# B&R Automation Studio project OpcUaSample410_BrbLibUa103 (part 13)

#### BrbUaRcGetNodeHandle.c
```c
#include <bur/plctypes.h>
#ifdef __cplusplus
	extern "C"
	{
#endif

#include "BrbLibUa.h"
#include <string.h>
#include <AnsiCFunc.h>

#ifdef __cplusplus
	};
#endif

// NOLINTBEGIN(readability-*, bugprone-easily-swappable-parameters, bugprone-branch-clone, clang-diagnostic-invalid-utf8, clang-diagnostic-invalid-source-encoding, clang-diagnostic-pointer-arith, clang-diagnostic-strict-prototypes, hicpp-uppercase-literal-suffix, cppcoreguidelines-*, performance-*)

/* Gibt einen ermittelten NodeHandle zurück */
unsigned short BrbUaRcGetNodeHandle(struct BrbUaRunClient_TYP* pRunClient, unsigned short nNodeHandleIndex, struct BrbUaRcNodeHandle_TYP* pNodeHandle)
{
	UINT nStatus = eBRB_ERR_NULL_POINTER;
	if(pRunClient != 0 && pNodeHandle != 0)
	{
		memset(pNodeHandle, 0, sizeof(BrbUaRcNodeHandle_TYP));
		nStatus = eBRB_ERR_UA_NO_ELEMENTS;
		if(pRunClient->NodeHandles.nNodeHandleCount > 0 && pRunClient->NodeHandles.pDatObjNamespaceIndices != 0 && pRunClient->NodeHandles.pNodeIds != 0 && pRunClient->NodeHandles.pNodeHandleErrorIds != 0 && pRunClient->NodeHandles.pNodeHandles != 0)
		{
			nStatus = eBRB_ERR_UA_INVALID_INDEX;
			if(nNodeHandleIndex < pRunClient->NodeHandles.nNodeHandleCount)
			{
				nStatus = eBRB_ERR_OK;
				pNodeHandle->nDatObjNamespaceIndex = *(((UINT*)pRunClient->NodeHandles.pDatObjNamespaceIndices) + nNodeHandleIndex);
				memcpy(&pNodeHandle->NodeId, (USINT*)(((UANodeID*)pRunClient->NodeHandles.pNodeIds) + nNodeHandleIndex), sizeof(UANodeID));
				pNodeHandle->nErrorId = *(((DWORD*)pRunClient->NodeHandles.pNodeHandleErrorIds) + nNodeHandleIndex);
				pNodeHandle->nNodeHandle = *(((DWORD*)pRunClient->NodeHandles.pNodeHandles) + nNodeHandleIndex);
			}
		}
	}
	return nStatus;
}

// NOLINTEND(readability-*, bugprone-easily-swappable-parameters, bugprone-branch-clone, clang-diagnostic-invalid-utf8, clang-diagnostic-invalid-source-encoding, clang-diagnostic-pointer-arith, clang-diagnostic-strict-prototypes, hicpp-uppercase-literal-suffix, cppcoreguidelines-*, performance-*)
```

#### BrbUaRcGetReadBlock.c
```c
#include <bur/plctypes.h>
#ifdef __cplusplus
	extern "C"
	{
#endif

#include "BrbLibUa.h"
#include <string.h>
#include <AnsiCFunc.h>

#ifdef __cplusplus
	};
#endif

// NOLINTBEGIN(readability-*, bugprone-easily-swappable-parameters, bugprone-branch-clone, clang-diagnostic-invalid-utf8, clang-diagnostic-invalid-source-encoding, clang-diagnostic-pointer-arith, clang-diagnostic-strict-prototypes, hicpp-uppercase-literal-suffix, cppcoreguidelines-*, performance-*)

/* Gibt einen ermittelten ReadBlock zurück */
unsigned short BrbUaRcGetReadBlock(struct BrbUaRunClient_TYP* pRunClient, unsigned short nReadBlockIndex, struct BrbUaRcReadBlock_TYP* pReadBlock, struct BrbUaRcReadBlockIntern_TYP* pReadBlockIntern)
{
	UINT nStatus = eBRB_ERR_NULL_POINTER;
	if(pRunClient != 0 && pReadBlock != 0)
	{
		memset(pReadBlock, 0, sizeof(BrbUaRcReadBlock_TYP));
		nStatus = eBRB_ERR_UA_NO_ELEMENTS;
		if(pRunClient->ReadBlocks.nBlockCount > 0 && pRunClient->ReadBlocks.pBlocks != 0)
		{
			nStatus = eBRB_ERR_UA_INVALID_INDEX;
			if(nReadBlockIndex < pRunClient->ReadBlocks.nBlockCount)
			{
				nStatus = eBRB_ERR_OK;
				BrbUaRcReadBlockIntern_TYP* pReadBlockInternOri = ((BrbUaRcReadBlockIntern_TYP*)pRunClient->ReadBlocks.pBlocks) + nReadBlockIndex;
				pReadBlock->nReadItemCount = pReadBlockInternOri->nReadItemCount;
				if(pReadBlockIntern != 0)
				{
					memcpy(pReadBlockIntern, pReadBlockInternOri, sizeof(BrbUaRcReadBlockIntern_TYP));
				}
			}
		}
	}
	return nStatus;
}

// NOLINTEND(readability-*, bugprone-easily-swappable-parameters, bugprone-branch-clone, clang-diagnostic-invalid-utf8, clang-diagnostic-invalid-source-encoding, clang-diagnostic-pointer-arith, clang-diagnostic-strict-prototypes, hicpp-uppercase-literal-suffix, cppcoreguidelines-*, performance-*)
```

#### BrbUaRcGetReadItem.c
```c
#include <bur/plctypes.h>
#ifdef __cplusplus
	extern "C"
	{
#endif

#include "BrbLibUa.h"
#include <string.h>
#include <AnsiCFunc.h>

#ifdef __cplusplus
	};
#endif

// NOLINTBEGIN(readability-*, bugprone-easily-swappable-parameters, bugprone-branch-clone, clang-diagnostic-invalid-utf8, clang-diagnostic-invalid-source-encoding, clang-diagnostic-pointer-arith, clang-diagnostic-strict-prototypes, hicpp-uppercase-literal-suffix, cppcoreguidelines-*, performance-*)

/* Gibt ein ermitteltes ReadItem zurück */
unsigned short BrbUaRcGetReadItem(struct BrbUaRunClient_TYP* pRunClient, unsigned short nReadBlockIndex, unsigned short nReadItemIndex, struct BrbUaRcReadItem_TYP* pReadItem)
{
	UINT nStatus = eBRB_ERR_NULL_POINTER;
	if(pRunClient != 0 && pReadItem != 0)
	{
		memset(pReadItem, 0, sizeof(BrbUaRcReadItem_TYP));
		nStatus = eBRB_ERR_UA_NO_ELEMENTS;
		if(pRunClient->ReadBlocks.nBlockCount > 0 && pRunClient->ReadBlocks.pBlocks != 0)
		{
			nStatus = eBRB_ERR_UA_INVALID_INDEX;
			if(nReadBlockIndex < pRunClient->ReadBlocks.nBlockCount)
			{
				nStatus = eBRB_ERR_UA_NO_ELEMENTS;
				BrbUaRcReadBlockIntern_TYP* pReadBlock = ((BrbUaRcReadBlockIntern_TYP*)pRunClient->ReadBlocks.pBlocks) + nReadBlockIndex;
				if(pReadBlock->nReadItemCount > 0 &&
					pReadBlock->pRiDatObjNamespaceIndices != 0 && pReadBlock->pRiNodeIds != 0 &&
					pReadBlock->pRiNodeAddInfos != 0 && pReadBlock->pRiVariables != 0 &&
					pReadBlock->pRiNodeErrorIds != 0 && pReadBlock->pRiTimestamps != 0
					)
				{
					nStatus = eBRB_ERR_UA_INVALID_INDEX;
					if(nReadItemIndex < pReadBlock->nReadItemCount)
					{
						nStatus = eBRB_ERR_OK;
						pReadItem->nDatObjNamespaceIndex = *(((UINT*)pReadBlock->pRiDatObjNamespaceIndices) + nReadItemIndex);
						memcpy(&pReadItem->NodeId, ((UANodeID*)pReadBlock->pRiNodeIds) + nReadItemIndex, sizeof(UANodeID));
						UANodeAdditionalInfo* pNodeAddInfo = ((UANodeAdditionalInfo*)pReadBlock->pRiNodeAddInfos) + nReadItemIndex;
						memcpy(&pReadItem->AddInfo, pNodeAddInfo, sizeof(UANodeAdditionalInfo));
						STRING sVarName[nBRBUA_VARNAME_TEXT_CHAR_MAX+1];
						STRING* pVar = (STRING*)((USINT*)pReadBlock->pRiVariables) + (nReadItemIndex * sizeof(sVarName));
						BrbStringCopy(pReadItem->sVar, pVar, sizeof(pReadItem->sVar));
						pReadItem->dtTimestamp = *(((DATE_AND_TIME*)pReadBlock->pRiTimestamps) + nReadItemIndex);
						pReadItem->nErrorId = *(((DWORD*)pReadBlock->pRiNodeErrorIds) + nReadItemIndex);
					}
				}
			}
		}
	}
	return nStatus;
}

// NOLINTEND(readability-*, bugprone-easily-swappable-parameters, bugprone-branch-clone, clang-diagnostic-invalid-utf8, clang-diagnostic-invalid-source-encoding, clang-diagnostic-pointer-arith, clang-diagnostic-strict-prototypes, hicpp-uppercase-literal-suffix, cppcoreguidelines-*, performance-*)
```

#### BrbUaRcGetWriteBlock.c
```c
#include <bur/plctypes.h>
#ifdef __cplusplus
	extern "C"
	{
#endif

#include "BrbLibUa.h"
#include <string.h>
#include <AnsiCFunc.h>

#ifdef __cplusplus
	};
#endif

// NOLINTBEGIN(readability-*, bugprone-easily-swappable-parameters, bugprone-branch-clone, clang-diagnostic-invalid-utf8, clang-diagnostic-invalid-source-encoding, clang-diagnostic-pointer-arith, clang-diagnostic-strict-prototypes, hicpp-uppercase-literal-suffix, cppcoreguidelines-*, performance-*)

/* Gibt einen ermittelten WriteBlock zurück */
unsigned short BrbUaRcGetWriteBlock(struct BrbUaRunClient_TYP* pRunClient, unsigned short nWriteBlockIndex, struct BrbUaRcWriteBlock_TYP* pWriteBlock, struct BrbUaRcWriteBlockIntern_TYP* pWriteBlockIntern)
{
	UINT nStatus = eBRB_ERR_NULL_POINTER;
	if(pRunClient != 0 && pWriteBlock != 0)
	{
		memset(pWriteBlock, 0, sizeof(BrbUaRcWriteBlock_TYP));
		nStatus = eBRB_ERR_UA_NO_ELEMENTS;
		if(pRunClient->WriteBlocks.nBlockCount > 0 && pRunClient->WriteBlocks.pBlocks != 0)
		{
			nStatus = eBRB_ERR_UA_INVALID_INDEX;
			if(nWriteBlockIndex < pRunClient->WriteBlocks.nBlockCount)
			{
				nStatus = eBRB_ERR_OK;
				BrbUaRcWriteBlockIntern_TYP* pWriteBlockInternOri = ((BrbUaRcWriteBlockIntern_TYP*)pRunClient->WriteBlocks.pBlocks) + nWriteBlockIndex;
				pWriteBlock->nWriteItemCount = pWriteBlockInternOri->nWriteItemCount;
				if(pWriteBlockIntern != 0)
				{
					memcpy(pWriteBlockIntern, pWriteBlockInternOri, sizeof(BrbUaRcWriteBlockIntern_TYP));
				}
			}
		}
	}
	return nStatus;
}

// NOLINTEND(readability-*, bugprone-easily-swappable-parameters, bugprone-branch-clone, clang-diagnostic-invalid-utf8, clang-diagnostic-invalid-source-encoding, clang-diagnostic-pointer-arith, clang-diagnostic-strict-prototypes, hicpp-uppercase-literal-suffix, cppcoreguidelines-*, performance-*)
```

#### BrbUaRcGetWriteItem.c
```c
#include <bur/plctypes.h>
#ifdef __cplusplus
	extern "C"
	{
#endif

#include "BrbLibUa.h"
#include <string.h>
#include <AnsiCFunc.h>

#ifdef __cplusplus
	};
#endif

// NOLINTBEGIN(readability-*, bugprone-easily-swappable-parameters, bugprone-branch-clone, clang-diagnostic-invalid-utf8, clang-diagnostic-invalid-source-encoding, clang-diagnostic-pointer-arith, clang-diagnostic-strict-prototypes, hicpp-uppercase-literal-suffix, cppcoreguidelines-*, performance-*)

/* Gibt ein ermitteltes WriteItem zurück */
unsigned short BrbUaRcGetWriteItem(struct BrbUaRunClient_TYP* pRunClient, unsigned short nWriteBlockIndex, unsigned short nWriteItemIndex, struct BrbUaRcWriteItem_TYP* pWriteItem)
{
	UINT nStatus = eBRB_ERR_NULL_POINTER;
	if(pRunClient != 0 && pWriteItem != 0)
	{
		memset(pWriteItem, 0, sizeof(BrbUaRcWriteItem_TYP));
		nStatus = eBRB_ERR_UA_NO_ELEMENTS;
		if(pRunClient->WriteBlocks.nBlockCount > 0 && pRunClient->WriteBlocks.pBlocks != 0)
		{
			nStatus = eBRB_ERR_UA_INVALID_INDEX;
			if(nWriteBlockIndex < pRunClient->WriteBlocks.nBlockCount)
			{
				nStatus = eBRB_ERR_UA_NO_ELEMENTS;
				BrbUaRcWriteBlockIntern_TYP* pWriteBlock = ((BrbUaRcWriteBlockIntern_TYP*)pRunClient->WriteBlocks.pBlocks) + nWriteBlockIndex;
				if(pWriteBlock->nWriteItemCount > 0 &&
					pWriteBlock->pWiDatObjNamespaceIndices != 0 && pWriteBlock->pWiNodeIds != 0 &&
					pWriteBlock->pWiNodeAddInfos != 0 && pWriteBlock->pWiVariables != 0 &&
					pWriteBlock->pWiNodeErrorIds != 0
					)
				{
					nStatus = eBRB_ERR_UA_INVALID_INDEX;
					if(nWriteItemIndex < pWriteBlock->nWriteItemCount)
					{
						nStatus = eBRB_ERR_OK;
						pWriteItem->nDatObjNamespaceIndex = *(((UINT*)pWriteBlock->pWiDatObjNamespaceIndices) + nWriteItemIndex);
						memcpy(&pWriteItem->NodeId, ((UANodeID*)pWriteBlock->pWiNodeIds) + nWriteItemIndex, sizeof(UANodeID));
						UANodeAdditionalInfo* pNodeAddInfo = ((UANodeAdditionalInfo*)pWriteBlock->pWiNodeAddInfos) + nWriteItemIndex;
						memcpy(&pWriteItem->AddInfo, pNodeAddInfo, sizeof(UANodeAdditionalInfo));
						STRING sVarName[nBRBUA_VARNAME_TEXT_CHAR_MAX+1];
						STRING* pVar = (STRING*)((USINT*)pWriteBlock->pWiVariables) + (nWriteItemIndex * sizeof(sVarName));
						BrbStringCopy(pWriteItem->sVar, pVar, sizeof(pWriteItem->sVar));
						pWriteItem->nErrorId = *(((DWORD*)pWriteBlock->pWiNodeErrorIds) + nWriteItemIndex);
					}
				}
			}
		}
	}
	return nStatus;
}

// NOLINTEND(readability-*, bugprone-easily-swappable-parameters, bugprone-branch-clone, clang-diagnostic-invalid-utf8, clang-diagnostic-invalid-source-encoding, clang-diagnostic-pointer-arith, clang-diagnostic-strict-prototypes, hicpp-uppercase-literal-suffix, cppcoreguidelines-*, performance-*)
```

#### BrbUaRcGetMethod.c
```c
#include <bur/plctypes.h>
#ifdef __cplusplus
	extern "C"
	{
#endif

#include "BrbLibUa.h"
#include <string.h>
#include <AnsiCFunc.h>

#ifdef __cplusplus
	};
#endif

// NOLINTBEGIN(readability-*, bugprone-easily-swappable-parameters, bugprone-branch-clone, clang-diagnostic-invalid-utf8, clang-diagnostic-invalid-source-encoding, clang-diagnostic-pointer-arith, clang-diagnostic-strict-prototypes, hicpp-uppercase-literal-suffix, cppcoreguidelines-*, performance-*)

/* Gibt eine ermittelte Methode zuück */
unsigned short BrbUaRcGetMethod(struct BrbUaRunClient_TYP* pRunClient, unsigned short nMethodIndex, struct BrbUaRcMethod_TYP* pMethod, struct BrbUaRcMethodIntern_TYP* pMethodIntern)
{
	UINT nStatus = eBRB_ERR_NULL_POINTER;
	if(pRunClient != 0 && pMethod != 0)
	{
		memset(pMethod, 0, sizeof(BrbUaRcMethod_TYP));
		nStatus = eBRB_ERR_UA_NO_ELEMENTS;
		if(pRunClient->Methods.nMethodCount > 0 && pRunClient->Methods.pMethods != 0)
		{
			nStatus = eBRB_ERR_UA_INVALID_INDEX;
			if(nMethodIndex < pRunClient->Methods.nMethodCount)
			{
				nStatus = eBRB_ERR_OK;
				BrbUaRcMethodIntern_TYP* pMethodInternOri = (((BrbUaRcMethodIntern_TYP*)pRunClient->Methods.pMethods)  + nMethodIndex);
				pMethod->nDatObjNamespaceIndex = pMethodInternOri->nDatObjNamespaceIndex;
				memcpy(&pMethod->ObjectNodeId, &pMethodInternOri->ObjectNodeId, sizeof(UANodeID));
				memcpy(&pMethod->MethodNodeId, &pMethodInternOri->MethodNodeId, sizeof(UANodeID));
				pMethod->tTimeout = pMethodInternOri->tTimeout;
				pMethod->nInputArgsCount = pMethodInternOri->nInputArgsCount;
				pMethod->nOutputArgsCount = pMethodInternOri->nOutputArgsCount;
				pMethod->nErrorId = pMethodInternOri->nErrorId;
				pMethod->nMethodHandle = pMethodInternOri->nMethodHandle;
				if(pMethodIntern != 0)
				{
					memcpy(pMethodIntern, pMethodInternOri, sizeof(BrbUaRcMethodIntern_TYP));
				}
			}
		}
	}
	return nStatus;
}

// NOLINTEND(readability-*, bugprone-easily-swappable-parameters, bugprone-branch-clone, clang-diagnostic-invalid-utf8, clang-diagnostic-invalid-source-encoding, clang-diagnostic-pointer-arith, clang-diagnostic-strict-prototypes, hicpp-uppercase-literal-suffix, cppcoreguidelines-*, performance-*)
```

#### BrbUaRcGetArgument.c
```c
#include <bur/plctypes.h>
#ifdef __cplusplus
	extern "C"
	{
#endif

#include "BrbLibUa.h"
#include <string.h>
#include <AnsiCFunc.h>

#ifdef __cplusplus
	};
#endif

// NOLINTBEGIN(readability-*, bugprone-easily-swappable-parameters, bugprone-branch-clone, clang-diagnostic-invalid-utf8, clang-diagnostic-invalid-source-encoding, clang-diagnostic-pointer-arith, clang-diagnostic-strict-prototypes, hicpp-uppercase-literal-suffix, cppcoreguidelines-*, performance-*)

/* Gibt ein ermitteltes ReadItem zurück */
unsigned short BrbUaRcGetArgument(struct BrbUaRunClient_TYP* pRunClient, unsigned short nMethodIndex, plcbit bOutput, unsigned short nArgumentIndex, struct UAMethodArgument* pArgument)
{
	UINT nStatus = eBRB_ERR_NULL_POINTER;
	if(pRunClient != 0 && pArgument != 0)
	{
		memset(pArgument, 0, sizeof(UAMethodArgument));
		nStatus = eBRB_ERR_UA_NO_ELEMENTS;
		if(pRunClient->Methods.nMethodCount > 0 && pRunClient->Methods.pMethods != 0)
		{
			nStatus = eBRB_ERR_UA_INVALID_INDEX;
			if(nMethodIndex < pRunClient->Methods.nMethodCount)
			{
				nStatus = eBRB_ERR_UA_NO_ELEMENTS;
				BrbUaRcMethodIntern_TYP* pMethod = (((BrbUaRcMethodIntern_TYP*)pRunClient->Methods.pMethods) + nMethodIndex);
				if(bOutput == 0)
				{
					if(pMethod->nInputArgsCount > 0 && pMethod->pInputArguments != 0)
					{
						nStatus = eBRB_ERR_UA_INVALID_INDEX;
						if(nArgumentIndex < pMethod->nInputArgsCount)
						{
							nStatus = eBRB_ERR_OK;
							UAMethodArgument* pArgumentIntern = ((UAMethodArgument*)pMethod->pInputArguments) + nArgumentIndex;
							memcpy(pArgument, pArgumentIntern, sizeof(UAMethodArgument));
						}
					}
				}
				else
				{
					if(pMethod->nOutputArgsCount > 0 && pMethod->pOutputArguments != 0)
					{
						nStatus = eBRB_ERR_UA_INVALID_INDEX;
						if(nArgumentIndex < pMethod->nOutputArgsCount)
						{
							nStatus = eBRB_ERR_OK;
							UAMethodArgument* pArgumentIntern = ((UAMethodArgument*)pMethod->pOutputArguments) + nArgumentIndex;
							memcpy(pArgument, pArgumentIntern, sizeof(UAMethodArgument));
						}
					}
				}
			}
		}
	}
	return nStatus;
}

// NOLINTEND(readability-*, bugprone-easily-swappable-parameters, bugprone-branch-clone, clang-diagnostic-invalid-utf8, clang-diagnostic-invalid-source-encoding, clang-diagnostic-pointer-arith, clang-diagnostic-strict-prototypes, hicpp-uppercase-literal-suffix, cppcoreguidelines-*, performance-*)
```

#### BrbUaRcGetSubscription.c
```c
#include <bur/plctypes.h>
#ifdef __cplusplus
	extern "C"
	{
#endif

#include "BrbLibUa.h"
#include <string.h>
#include <AnsiCFunc.h>

#ifdef __cplusplus
	};
#endif

// NOLINTBEGIN(readability-*, bugprone-easily-swappable-parameters, bugprone-branch-clone, clang-diagnostic-invalid-utf8, clang-diagnostic-invalid-source-encoding, clang-diagnostic-pointer-arith, clang-diagnostic-strict-prototypes, hicpp-uppercase-literal-suffix, cppcoreguidelines-*, performance-*)

/* Gibt eine ermittelte Subscription zurück */
unsigned short BrbUaRcGetSubscription(struct BrbUaRunClient_TYP* pRunClient, unsigned short nSubscriptionIndex, struct BrbUaRcSubscription_TYP* pSubscription, struct BrbUaRcSubscriptionIntern_TYP* pSubscriptionIntern)
{
	UINT nStatus = eBRB_ERR_NULL_POINTER;
	if(pRunClient != 0 && pSubscription != 0)
	{
		memset(pSubscription, 0, sizeof(BrbUaRcSubscription_TYP));
		nStatus = eBRB_ERR_UA_NO_ELEMENTS;
		if(pRunClient->Subscriptions.nSubscriptionCount > 0 && pRunClient->Subscriptions.pSubscriptions != 0)
		{
			nStatus = eBRB_ERR_UA_INVALID_INDEX;
			if(nSubscriptionIndex < pRunClient->Subscriptions.nSubscriptionCount)
			{
				nStatus = eBRB_ERR_OK;
				BrbUaRcSubscriptionIntern_TYP* pSubscriptionInternOri = ((BrbUaRcSubscriptionIntern_TYP*)pRunClient->Subscriptions.pSubscriptions) + nSubscriptionIndex;
				pSubscription->bPublishingEnable = pSubscriptionInternOri->bPublishingEnable;
				pSubscription->nPriority = pSubscriptionInternOri->nPriority;
				pSubscription->tPublishingInterval = pSubscriptionInternOri->tPublishingInterval;
				pSubscription->nMonitoredItemCount = pSubscriptionInternOri->nMonitoredItemCount;
				pSubscription->nEventItemCount = pSubscriptionInternOri->nEventItemCount;
				pSubscription->nErrorId = pSubscriptionInternOri->nErrorId;
				pSubscription->nSubscriptionHandle = pSubscriptionInternOri->nSubscriptionHandle;
				if(pSubscriptionIntern != 0)
				{
					memcpy(pSubscriptionIntern, pSubscriptionInternOri, sizeof(BrbUaRcSubscriptionIntern_TYP));
				}
			}
		}
	}
	return nStatus;
}

// NOLINTEND(readability-*, bugprone-easily-swappable-parameters, bugprone-branch-clone, clang-diagnostic-invalid-utf8, clang-diagnostic-invalid-source-encoding, clang-diagnostic-pointer-arith, clang-diagnostic-strict-prototypes, hicpp-uppercase-literal-suffix, cppcoreguidelines-*, performance-*)
```

#### BrbUaRcSetSubscription.c
```c
#include <bur/plctypes.h>
#ifdef __cplusplus
	extern "C"
	{
#endif

#include "BrbLibUa.h"
#include <string.h>
#include <AnsiCFunc.h>

#ifdef __cplusplus
	};
#endif

// NOLINTBEGIN(readability-*, bugprone-easily-swappable-parameters, bugprone-branch-clone, clang-diagnostic-invalid-utf8, clang-diagnostic-invalid-source-encoding, clang-diagnostic-pointer-arith, clang-diagnostic-strict-prototypes, hicpp-uppercase-literal-suffix, cppcoreguidelines-*, performance-*)

// Eigene Enums und Typen
enum Steps_ENUM
{
	eSTEP_INIT,
	eSTEP_OPERATE,
	eSTEP_OPERATE_WAIT,
};

/* Ändert die Parameter einer Subscription */
void BrbUaRcSetSubscription(struct BrbUaRcSetSubscription* inst)
{
	switch(inst->eStep)
	{
		case eSTEP_INIT:
			// Fub initialisieren
			inst->nStatus =  eBRB_ERR_BUSY;
			inst->bPublished = 0;
			inst->nErrorId = 0x00000000; // Good
			BrbUaGetStatusCodeText(inst->nErrorId, inst->sErrorId, sizeof(inst->nErrorId));
			memset(&inst->fbUA_SubscriptionOperate, 0, sizeof(inst->fbUA_SubscriptionOperate));
			// Parameter prüfen
			if(inst->pRunClient != 0 && inst->pSubscription != 0)
			{
				if(inst->pRunClient->State.eClientState == eBRB_RCCLTSTATE_CONNECTED && inst->pRunClient->Connection.nConnectionHandle != 0)
				{
					if(inst->pRunClient->Subscriptions.nSubscriptionCount > 0 && inst->pRunClient->Subscriptions.pSubscriptions != 0)
					{
						if(inst->nSubscriptionIndex < inst->pRunClient->Subscriptions.nSubscriptionCount)
						{
							inst->eStep = eSTEP_OPERATE;
						}
						else
						{
							inst->nStatus = eBRB_ERR_UA_INVALID_INDEX;
						}
					}
					else
					{
						inst->nStatus = eBRB_ERR_UA_NO_ELEMENTS;
					}
				}
				else
				{
					inst->nStatus = eBRB_ERR_UA_NOT_CONNECTED;
				}
			}
			else
			{
				inst->nStatus = eBRB_ERR_NULL_POINTER;
			}
			break;

		case eSTEP_OPERATE:
			// Subscription ändern
			inst->nStatus  = eBRB_ERR_BUSY;
			{
				BrbUaRcSubscriptionIntern_TYP* pSubscriptionIntern = ((BrbUaRcSubscriptionIntern_TYP*)inst->pRunClient->Subscriptions.pSubscriptions) + inst->nSubscriptionIndex;
				inst->fbUA_SubscriptionOperate.Execute = 1;
				inst->fbUA_SubscriptionOperate.SubscriptionHdl = pSubscriptionIntern->nSubscriptionHandle;
				inst->fbUA_SubscriptionOperate.PublishingEnable = inst->pSubscription->bPublishingEnable;
				inst->fbUA_SubscriptionOperate.Priority = inst->pSubscription->nPriority;
				inst->fbUA_SubscriptionOperate.Timeout = inst->pRunClient->Cfg.tAccessTimeout;
				inst->tPublishingInterval = inst->pSubscription->tPublishingInterval;
				inst->fbUA_SubscriptionOperate.PublishingInterval = &inst->tPublishingInterval;
			}
			inst->eStep = eSTEP_OPERATE_WAIT;
			break;

		case eSTEP_OPERATE_WAIT:
			// Warten, bis Subscription geändert wurde
			inst->nStatus  = eBRB_ERR_BUSY;
			if(inst->fbUA_SubscriptionOperate.Done == 1)
			{
				inst->fbUA_SubscriptionOperate.Execute = 0;
				// Geänderte Werte in interne Daten übernehmen
				BrbUaRcSubscriptionIntern_TYP* pSubscriptionIntern = ((BrbUaRcSubscriptionIntern_TYP*)inst->pRunClient->Subscriptions.pSubscriptions) + inst->nSubscriptionIndex;
				pSubscriptionIntern->bPublishingEnable = inst->pSubscription->bPublishingEnable;
				pSubscriptionIntern->nPriority = inst->pSubscription->nPriority;
				pSubscriptionIntern->tPublishingInterval = inst->pSubscription->tPublishingInterval = inst->tPublishingInterval;
				inst->nStatus  = eBRB_ERR_OK;
				inst->bPublished = inst->fbUA_SubscriptionOperate.Published;
				inst->nErrorId = inst->fbUA_SubscriptionOperate.ErrorID;
				BrbUaGetStatusCodeText(inst->nErrorId, inst->sErrorId, sizeof(inst->nErrorId));
				inst->eStep = eSTEP_INIT;
			}
			else if(inst->fbUA_SubscriptionOperate.Error == 1)
			{
				inst->fbUA_SubscriptionOperate.Execute = 0;
				inst->nStatus  = eBRB_ERR_UA_ERROR;
				inst->nErrorId = inst->fbUA_SubscriptionOperate.ErrorID;
				BrbUaGetStatusCodeText(inst->nErrorId, inst->sErrorId, sizeof(inst->nErrorId));
				inst->eStep = eSTEP_INIT;
			}
			break;

	}

	// Aufruf aller FB's
	UA_SubscriptionOperate(&inst->fbUA_SubscriptionOperate);

}

// NOLINTEND(readability-*, bugprone-easily-swappable-parameters, bugprone-branch-clone, clang-diagnostic-invalid-utf8, clang-diagnostic-invalid-source-encoding, clang-diagnostic-pointer-arith, clang-diagnostic-strict-prototypes, hicpp-uppercase-literal-suffix, cppcoreguidelines-*, performance-*)
```

#### BrbUaRcGetMonitoredItem.c
```c
#include <bur/plctypes.h>
#ifdef __cplusplus
	extern "C"
	{
#endif

#include "BrbLibUa.h"
#include <string.h>
#include <AnsiCFunc.h>

#ifdef __cplusplus
	};
#endif

// NOLINTBEGIN(readability-*, bugprone-easily-swappable-parameters, bugprone-branch-clone, clang-diagnostic-invalid-utf8, clang-diagnostic-invalid-source-encoding, clang-diagnostic-pointer-arith, clang-diagnostic-strict-prototypes, hicpp-uppercase-literal-suffix, cppcoreguidelines-*, performance-*)

/* Gibt ein ermitteltes MonitoredItem zurück */
unsigned short BrbUaRcGetMonitoredItem(struct BrbUaRunClient_TYP* pRunClient, unsigned short nSubscriptionIndex, unsigned short nMonitoredItemIndex, struct BrbUaRcMonitoredItem_TYP* pMonitoredItem)
{
	UINT nStatus = eBRB_ERR_NULL_POINTER;
	if(pRunClient != 0 && pMonitoredItem != 0)
	{
		memset(pMonitoredItem, 0, sizeof(BrbUaRcMonitoredItem_TYP));
		nStatus = eBRB_ERR_UA_NO_ELEMENTS;
		if(pRunClient->Subscriptions.nSubscriptionCount > 0 && pRunClient->Subscriptions.pSubscriptions != 0)
		{
			nStatus = eBRB_ERR_UA_INVALID_INDEX;
			if(nSubscriptionIndex < pRunClient->Subscriptions.nSubscriptionCount)
			{
				nStatus = eBRB_ERR_UA_NO_ELEMENTS;
				BrbUaRcSubscriptionIntern_TYP* pSubscription = ((BrbUaRcSubscriptionIntern_TYP*)pRunClient->Subscriptions.pSubscriptions) + nSubscriptionIndex;
				if(pSubscription->nMonitoredItemCount > 0 &&
					pSubscription->pMiDatObjNamespaceIndices != 0 && pSubscription->pMiNodeIds != 0 &&
					pSubscription->pMiNodeHandleErrorIds != 0 && pSubscription->pMiNodeHandles != 0 &&
					pSubscription->pMiNodeAddInfos != 0 && pSubscription->pMiVariables != 0 &&
					pSubscription->pMiQueueSizeOri != 0 && pSubscription->pMiMonitorSettings != 0 &&
					pSubscription->pMiValuesChanged != 0 && pSubscription->pMiRemainingValueCounts != 0 &&
					pSubscription->pMiTimestamps != 0 && pSubscription->pMiNodeQualityIds != 0 &&
					pSubscription->pMiMonitoredItemErrorIds != 0 && pSubscription->pMiMonitoredItemHandles != 0
					)
				{
					nStatus = eBRB_ERR_UA_INVALID_INDEX;
					if(nMonitoredItemIndex < pSubscription->nMonitoredItemCount)
					{
						nStatus = eBRB_ERR_OK;
						pMonitoredItem->nDatObjNamespaceIndex = *(((UINT*)pSubscription->pMiDatObjNamespaceIndices) + nMonitoredItemIndex);
						memcpy(&pMonitoredItem->NodeId, ((UANodeID*)pSubscription->pMiNodeIds) + nMonitoredItemIndex, sizeof(UANodeID));
						pMonitoredItem->nNodeHandleErrorId = *(((DWORD*)pSubscription->pMiNodeHandleErrorIds) + nMonitoredItemIndex);
						pMonitoredItem->nNodeHandle = *(((DWORD*)pSubscription->pMiNodeHandles) + nMonitoredItemIndex);
						UANodeAdditionalInfo* pNodeAddInfo = ((UANodeAdditionalInfo*)pSubscription->pMiNodeAddInfos) + nMonitoredItemIndex;
						memcpy(&pMonitoredItem->AddInfo, pNodeAddInfo, sizeof(UANodeAdditionalInfo));
						STRING sVarName[nBRBUA_VARNAME_TEXT_CHAR_MAX+1];
						STRING* pVar = (STRING*)((USINT*)pSubscription->pMiVariables) + (nMonitoredItemIndex * sizeof(sVarName));
						BrbStringCopy(pMonitoredItem->sVar, pVar, sizeof(pMonitoredItem->sVar));
						pMonitoredItem->nQueueSizeOri = *(((UINT*)pSubscription->pMiQueueSizeOri) + nMonitoredItemIndex);
						UAMonitoringParameters* pMonitoringSetting = ((UAMonitoringParameters*)pSubscription->pMiMonitorSettings) + nMonitoredItemIndex;
						memcpy(&pMonitoredItem->MonitorSettings, pMonitoringSetting, sizeof(UAMonitoringParameters));
						pMonitoredItem->bValueChanged = *(((BOOL*)pSubscription->pMiValuesChanged) + nMonitoredItemIndex);
						pMonitoredItem->nRemainingValueCount = *(((UINT*)pSubscription->pMiRemainingValueCounts) + nMonitoredItemIndex);
						pMonitoredItem->dtTimestamp = *(((DT*)pSubscription->pMiTimestamps) + nMonitoredItemIndex);
						pMonitoredItem->nNodeQualityId = *(((DWORD*)pSubscription->pMiNodeQualityIds) + nMonitoredItemIndex);
						pMonitoredItem->nMonitoredItemErrorId = *(((DWORD*)pSubscription->pMiMonitoredItemErrorIds) + nMonitoredItemIndex);
						pMonitoredItem->nMonitoredItemHandle = *(((DWORD*)pSubscription->pMiMonitoredItemHandles) + nMonitoredItemIndex);
					}
				}
			}
		}
	}
	return nStatus;
}

// NOLINTEND(readability-*, bugprone-easily-swappable-parameters, bugprone-branch-clone, clang-diagnostic-invalid-utf8, clang-diagnostic-invalid-source-encoding, clang-diagnostic-pointer-arith, clang-diagnostic-strict-prototypes, hicpp-uppercase-literal-suffix, cppcoreguidelines-*, performance-*)
```

#### BrbUaRcSetMonitoredItem.c
```c
#include <bur/plctypes.h>
#ifdef __cplusplus
	extern "C"
	{
#endif

#include "BrbLibUa.h"
#include <string.h>
#include <AnsiCFunc.h>

#ifdef __cplusplus
	};
#endif

// NOLINTBEGIN(readability-*, bugprone-easily-swappable-parameters, bugprone-branch-clone, clang-diagnostic-invalid-utf8, clang-diagnostic-invalid-source-encoding, clang-diagnostic-pointer-arith, clang-diagnostic-strict-prototypes, hicpp-uppercase-literal-suffix, cppcoreguidelines-*, performance-*)

// Eigene Enums und Typen
enum Steps_ENUM
{
	eSTEP_INIT,
	eSTEP_OPERATE,
	eSTEP_OPERATE_WAIT,
};

/* Ändert die Parameter eines MonitoredItems */
void BrbUaRcSetMonitoredItem(struct BrbUaRcSetMonitoredItem* inst)
{
	switch(inst->eStep)
	{
		case eSTEP_INIT:
			// Fub initialisieren
			inst->nStatus =  eBRB_ERR_BUSY;
			inst->bValueChanged = 0;
			inst->dtTimestamp = 0;
			inst->nErrorId = 0x00000000; // Good
			BrbUaGetStatusCodeText(inst->nErrorId, inst->sErrorId, sizeof(inst->nErrorId));
			memset(&inst->fbUA_MonitoredItemOperate, 0, sizeof(inst->fbUA_MonitoredItemOperate));
			// Parameter prüfen
			if(inst->pRunClient != 0 && inst->pMonitoringSettings != 0)
			{
				if(inst->pRunClient->State.eClientState == eBRB_RCCLTSTATE_CONNECTED && inst->pRunClient->Connection.nConnectionHandle != 0)
				{
					if(inst->pRunClient->Subscriptions.nSubscriptionCount > 0 && inst->pRunClient->Subscriptions.pSubscriptions != 0)
					{
						if(inst->nSubscriptionIndex < inst->pRunClient->Subscriptions.nSubscriptionCount)
						{
							BrbUaRcSubscriptionIntern_TYP* pSubscriptionIntern = ((BrbUaRcSubscriptionIntern_TYP*)inst->pRunClient->Subscriptions.pSubscriptions) + inst->nSubscriptionIndex;
							if(pSubscriptionIntern->nMonitoredItemCount > 0 &&
								pSubscriptionIntern->pMiDatObjNamespaceIndices != 0 && pSubscriptionIntern->pMiNodeIds != 0 &&
								pSubscriptionIntern->pMiNodeHandleErrorIds != 0 && pSubscriptionIntern->pMiNodeHandles != 0 &&
								pSubscriptionIntern->pMiNodeAddInfos != 0 && pSubscriptionIntern->pMiVariables != 0 &&
								pSubscriptionIntern->pMiQueueSizeOri != 0 && pSubscriptionIntern->pMiMonitorSettings != 0 &&
								pSubscriptionIntern->pMiValuesChanged != 0 && pSubscriptionIntern->pMiRemainingValueCounts != 0 &&
								pSubscriptionIntern->pMiTimestamps != 0 && pSubscriptionIntern->pMiNodeQualityIds != 0 &&
								pSubscriptionIntern->pMiMonitoredItemErrorIds != 0 && pSubscriptionIntern->pMiMonitoredItemHandles != 0)
							{
								if(inst->nMonitoredItemIndex < pSubscriptionIntern->nMonitoredItemCount)
								{
									inst->eStep = eSTEP_OPERATE;
								}
								else
								{
									inst->nStatus = eBRB_ERR_UA_INVALID_INDEX;
								}
							}
							else
							{
								inst->nStatus = eBRB_ERR_UA_NO_ELEMENTS;
							}
						}
						else
						{
							inst->nStatus = eBRB_ERR_UA_NOT_CONNECTED;
						}
					}
					else
					{
						inst->nStatus = eBRB_ERR_UA_NO_ELEMENTS;
					}
				}
				else
				{
					inst->nStatus = eBRB_ERR_UA_NOT_CONNECTED;
				}
			}
			else
			{
				inst->nStatus = eBRB_ERR_NULL_POINTER;
			}
			break;

		case eSTEP_OPERATE:
			// MonitoredItem ändern
			inst->nStatus  = eBRB_ERR_BUSY;
			BrbUaRcGetMonitoredItem(inst->pRunClient, inst->nSubscriptionIndex, inst->nMonitoredItemIndex, &inst->MonitoredItemIntern);
			inst->fbUA_MonitoredItemOperate.Execute = 1;
			inst->fbUA_MonitoredItemOperate.MonitoredItemHdl = inst->MonitoredItemIntern.nMonitoredItemHandle;
			inst->fbUA_MonitoredItemOperate.Timeout = inst->pRunClient->Cfg.tAccessTimeout;
			inst->fbUA_MonitoredItemOperate.MonitoringSettings = inst->pMonitoringSettings;
			inst->eStep = eSTEP_OPERATE_WAIT;
			break;

		case eSTEP_OPERATE_WAIT:
			// Warten, bis MonitoredItem geändert wurde
			inst->nStatus  = eBRB_ERR_BUSY;
			if(inst->fbUA_MonitoredItemOperate.Done == 1)
			{
				inst->fbUA_MonitoredItemOperate.Execute = 0;
				// Geänderte Werte in interne Daten übernehmen
				BrbUaRcSubscriptionIntern_TYP* pSubscriptionIntern = ((BrbUaRcSubscriptionIntern_TYP*)inst->pRunClient->Subscriptions.pSubscriptions) + inst->nSubscriptionIndex;
				UAMonitoringParameters* pMonitoringSettingIntern = ((UAMonitoringParameters*)pSubscriptionIntern->pMiMonitorSettings) + inst->nMonitoredItemIndex;
				pMonitoringSettingIntern->SamplingInterval = inst->pMonitoringSettings->SamplingInterval;
				pMonitoringSettingIntern->DeadbandType = inst->pMonitoringSettings->DeadbandType;
				pMonitoringSettingIntern->Deadband = inst->pMonitoringSettings->Deadband;
				inst->nStatus  = eBRB_ERR_OK;
				inst->bValueChanged = inst->fbUA_MonitoredItemOperate.ValueChanged;
				inst->dtTimestamp = inst->fbUA_MonitoredItemOperate.TimeStamp;
				inst->nErrorId = inst->fbUA_MonitoredItemOperate.ErrorID;
				BrbUaGetStatusCodeText(inst->nErrorId, inst->sErrorId, sizeof(inst->nErrorId));
				inst->eStep = eSTEP_INIT;
			}
			else if(inst->fbUA_MonitoredItemOperate.Error == 1)
			{
				inst->fbUA_MonitoredItemOperate.Execute = 0;
				inst->nStatus  = eBRB_ERR_UA_ERROR;
				inst->nErrorId = inst->fbUA_MonitoredItemOperate.ErrorID;
				BrbUaGetStatusCodeText(inst->nErrorId, inst->sErrorId, sizeof(inst->nErrorId));
				inst->eStep = eSTEP_INIT;
			}
			break;

	}

	// Aufruf aller FB's
	UA_MonitoredItemOperate(&inst->fbUA_MonitoredItemOperate);

}

// NOLINTEND(readability-*, bugprone-easily-swappable-parameters, bugprone-branch-clone, clang-diagnostic-invalid-utf8, clang-diagnostic-invalid-source-encoding, clang-diagnostic-pointer-arith, clang-diagnostic-strict-prototypes, hicpp-uppercase-literal-suffix, cppcoreguidelines-*, performance-*)
```

#### BrbUaRcGetMiValueChanged.c
```c
#include <bur/plctypes.h>
#ifdef __cplusplus
	extern "C"
	{
#endif

#include "BrbLibUa.h"
#include <string.h>
#include <AnsiCFunc.h>

#ifdef __cplusplus
	};
#endif

// NOLINTBEGIN(readability-*, bugprone-easily-swappable-parameters, bugprone-branch-clone, clang-diagnostic-invalid-utf8, clang-diagnostic-invalid-source-encoding, clang-diagnostic-pointer-arith, clang-diagnostic-strict-prototypes, hicpp-uppercase-literal-suffix, cppcoreguidelines-*, performance-*)

/* Gibt das ValueChanged-Flag eines MonitoredItems zurück und löscht es optional */
plcbit BrbUaRcGetMiValueChanged(struct BrbUaRunClient_TYP* pRunClient, unsigned short nSubscriptionIndex, unsigned short nMonitoredItemIndex, plcbit bClear)
{
	BOOL bResult = 0;
	if(pRunClient != 0)
	{
		if(pRunClient->State.eClientState == eBRB_RCCLTSTATE_CONNECTED)
		{
			if(pRunClient->Subscriptions.nSubscriptionCount > 0 &&pRunClient->Subscriptions.pSubscriptions != 0)
			{
				if(nSubscriptionIndex < pRunClient->Subscriptions.nSubscriptionCount)
				{
					BrbUaRcSubscriptionIntern_TYP* pSubscription = ((BrbUaRcSubscriptionIntern_TYP*)pRunClient->Subscriptions.pSubscriptions) + nSubscriptionIndex;
					if(pSubscription->nMonitoredItemCount > 0 &&
						pSubscription->pMiDatObjNamespaceIndices != 0 && pSubscription->pMiNodeIds != 0 &&
						pSubscription->pMiNodeHandleErrorIds != 0 && pSubscription->pMiNodeHandles != 0 &&
						pSubscription->pMiNodeAddInfos != 0 && pSubscription->pMiVariables != 0 &&
						pSubscription->pMiQueueSizeOri != 0 && pSubscription->pMiMonitorSettings != 0 &&
						pSubscription->pMiValuesChanged != 0 && pSubscription->pMiRemainingValueCounts != 0 &&
						pSubscription->pMiTimestamps != 0 && pSubscription->pMiNodeQualityIds != 0 &&
						pSubscription->pMiMonitoredItemErrorIds != 0 && pSubscription->pMiMonitoredItemHandles != 0)
					{
						if(nMonitoredItemIndex < pSubscription->nMonitoredItemCount)
						{
							bResult = *(((BOOL*)pSubscription->pMiValuesChanged) + nMonitoredItemIndex);
							if(bClear == 1)
							{
								*(((BOOL*)pSubscription->pMiValuesChanged) + nMonitoredItemIndex) = 0;
							}
						}
					}
				}
			}
		}
	}
	return bResult;
}

// NOLINTEND(readability-*, bugprone-easily-swappable-parameters, bugprone-branch-clone, clang-diagnostic-invalid-utf8, clang-diagnostic-invalid-source-encoding, clang-diagnostic-pointer-arith, clang-diagnostic-strict-prototypes, hicpp-uppercase-literal-suffix, cppcoreguidelines-*, performance-*)
```

#### BrbUaRcGetMiRemainingValueCount.c
```c
#include <bur/plctypes.h>
#ifdef __cplusplus
	extern "C"
	{
#endif

#include "BrbLibUa.h"
#include <string.h>
#include <AnsiCFunc.h>

#ifdef __cplusplus
	};
#endif

// NOLINTBEGIN(readability-*, bugprone-easily-swappable-parameters, bugprone-branch-clone, clang-diagnostic-invalid-utf8, clang-diagnostic-invalid-source-encoding, clang-diagnostic-pointer-arith, clang-diagnostic-strict-prototypes, hicpp-uppercase-literal-suffix, cppcoreguidelines-*, performance-*)

/* Gibt den RemainingValue-Zähler eines MonitoredItems zurück */
unsigned short BrbUaRcGetMiRemainingValueCount(struct BrbUaRunClient_TYP* pRunClient, unsigned short nSubscriptionIndex, unsigned short nMonitoredItemIndex)
{
	UINT nResult = 0;
	if(pRunClient != 0)
	{
		if(pRunClient->State.eClientState == eBRB_RCCLTSTATE_CONNECTED)
		{
			if(pRunClient->Subscriptions.nSubscriptionCount > 0 &&pRunClient->Subscriptions.pSubscriptions != 0)
			{
				if(nSubscriptionIndex < pRunClient->Subscriptions.nSubscriptionCount)
				{
					BrbUaRcSubscriptionIntern_TYP* pSubscription = ((BrbUaRcSubscriptionIntern_TYP*)pRunClient->Subscriptions.pSubscriptions) + nSubscriptionIndex;
					if(pSubscription->nMonitoredItemCount > 0 &&
						pSubscription->pMiDatObjNamespaceIndices != 0 && pSubscription->pMiNodeIds != 0 &&
						pSubscription->pMiNodeHandleErrorIds != 0 && pSubscription->pMiNodeHandles != 0 &&
						pSubscription->pMiNodeAddInfos != 0 && pSubscription->pMiVariables != 0 &&
						pSubscription->pMiQueueSizeOri != 0 && pSubscription->pMiMonitorSettings != 0 &&
						pSubscription->pMiValuesChanged != 0 && pSubscription->pMiRemainingValueCounts != 0 &&
						pSubscription->pMiTimestamps != 0 && pSubscription->pMiNodeQualityIds != 0 &&
						pSubscription->pMiMonitoredItemErrorIds != 0 && pSubscription->pMiMonitoredItemHandles != 0)
					{
						if(nMonitoredItemIndex < pSubscription->nMonitoredItemCount)
						{
							nResult = *(((UINT*)pSubscription->pMiRemainingValueCounts) + nMonitoredItemIndex);
						}
					}
				}
			}
		}
	}
	return nResult;
}

// NOLINTEND(readability-*, bugprone-easily-swappable-parameters, bugprone-branch-clone, clang-diagnostic-invalid-utf8, clang-diagnostic-invalid-source-encoding, clang-diagnostic-pointer-arith, clang-diagnostic-strict-prototypes, hicpp-uppercase-literal-suffix, cppcoreguidelines-*, performance-*)
```

#### BrbUaRcGetEventItem.c
```c
#include <bur/plctypes.h>
#ifdef __cplusplus
	extern "C"
	{
#endif

#include "BrbLibUa.h"
#include <string.h>
#include <AnsiCFunc.h>

#ifdef __cplusplus
	};
#endif

// NOLINTBEGIN(readability-*, bugprone-easily-swappable-parameters, bugprone-branch-clone, clang-diagnostic-invalid-utf8, clang-diagnostic-invalid-source-encoding, clang-diagnostic-pointer-arith, clang-diagnostic-strict-prototypes, hicpp-uppercase-literal-suffix, cppcoreguidelines-*, performance-*)

/* Gibt ein ermitteltes EventItem zurück */
unsigned short BrbUaRcGetEventItem(struct BrbUaRunClient_TYP* pRunClient, unsigned short nSubscriptionIndex, unsigned short nEventItemIndex, struct BrbUaRcEventItem_TYP* pEventItem, struct BrbUaRcEventItemIntern_TYP* pEventItemIntern)
{
	UINT nStatus = eBRB_ERR_NULL_POINTER;
	if(pRunClient != 0 && pEventItem != 0)
	{
		memset(pEventItem, 0, sizeof(BrbUaRcEventItem_TYP));
		nStatus = eBRB_ERR_UA_NO_ELEMENTS;
		if(pRunClient->Subscriptions.nSubscriptionCount > 0 && pRunClient->Subscriptions.pSubscriptions != 0)
		{
			nStatus = eBRB_ERR_UA_INVALID_INDEX;
			if(nSubscriptionIndex < pRunClient->Subscriptions.nSubscriptionCount)
			{
				nStatus = eBRB_ERR_UA_NO_ELEMENTS;
				BrbUaRcSubscriptionIntern_TYP* pSubscription = ((BrbUaRcSubscriptionIntern_TYP*)pRunClient->Subscriptions.pSubscriptions) + nSubscriptionIndex;
				if(pSubscription->nEventItemCount > 0 && pSubscription->pEventItems != 0)
				{
					nStatus = eBRB_ERR_UA_INVALID_INDEX;
					if(nEventItemIndex < pSubscription->nEventItemCount)
					{
						nStatus = eBRB_ERR_OK;
						BrbUaRcEventItemIntern_TYP* pEventItemInternOri = ((BrbUaRcEventItemIntern_TYP*)pSubscription->pEventItems) + nEventItemIndex;
						pEventItem->nEventDatObjNamespaceIndex = pEventItemInternOri->nEventDatObjNamespaceIndex;
						memcpy(&pEventItem->EventNodeId, &pEventItemInternOri->EventNodeId, sizeof(UANodeID));
						pEventItem->nEventNodeHandleErrorId = pEventItemInternOri->nEventNodeHandleErrorId;
						pEventItem->nEventNodeHandle = pEventItemInternOri->nEventNodeHandle;
						pEventItem->nTypeDatObjNamespaceIndex = pEventItemInternOri->nTypeDatObjNamespaceIndex;
						memcpy(&pEventItem->TypeNodeId, &pEventItemInternOri->TypeNodeId, sizeof(UANodeID));
						pEventItem->nEventItemErrorId = pEventItemInternOri->nEventItemErrorId;
						pEventItem->nEventItemHandle = pEventItemInternOri->nEventItemHandle;
						pEventItem->tTimeout = pEventItemInternOri->tTimeout;
						pEventItem->bCallOperate = pEventItemInternOri->bCallOperate;
						pEventItem->nEventFieldCount = pEventItemInternOri->nEventFieldCount;
						pEventItem->nReceiveCount = pEventItemInternOri->nReceiveCount;
						pEventItem->bEventReceived = pEventItemInternOri->bEventReceived;
						if(pEventItemIntern != 0)
						{
							memcpy(pEventItemIntern, pEventItemInternOri, sizeof(BrbUaRcEventItemIntern_TYP));
						}
					}
				}
			}
		}
	}
	return nStatus;
}

// NOLINTEND(readability-*, bugprone-easily-swappable-parameters, bugprone-branch-clone, clang-diagnostic-invalid-utf8, clang-diagnostic-invalid-source-encoding, clang-diagnostic-pointer-arith, clang-diagnostic-strict-prototypes, hicpp-uppercase-literal-suffix, cppcoreguidelines-*, performance-*)
```

#### BrbUaRcGetEventItemReceived.c
```c
#include <bur/plctypes.h>
#ifdef __cplusplus
	extern "C"
	{
#endif

#include "BrbLibUa.h"
#include <string.h>
#include <AnsiCFunc.h>

#ifdef __cplusplus
	};
#endif

// NOLINTBEGIN(readability-*, bugprone-easily-swappable-parameters, bugprone-branch-clone, clang-diagnostic-invalid-utf8, clang-diagnostic-invalid-source-encoding, clang-diagnostic-pointer-arith, clang-diagnostic-strict-prototypes, hicpp-uppercase-literal-suffix, cppcoreguidelines-*, performance-*)

/* Gibt zurück, ob ein Event empfangen wurde */
plcbit BrbUaRcGetEventItemReceived(struct BrbUaRunClient_TYP* pRunClient, unsigned short nSubscriptionIndex, unsigned short nEventItemIndex)
{
	BOOL bResult = 0;
	if(pRunClient != 0)
	{
		if(pRunClient->State.eClientState == eBRB_RCCLTSTATE_CONNECTED)
		{
			if(pRunClient->Subscriptions.nSubscriptionCount > 0 && pRunClient->Subscriptions.pSubscriptions != 0)
			{
				if(nSubscriptionIndex < pRunClient->Subscriptions.nSubscriptionCount)
				{
					BrbUaRcSubscriptionIntern_TYP* pSubscription = ((BrbUaRcSubscriptionIntern_TYP*)pRunClient->Subscriptions.pSubscriptions) + nSubscriptionIndex;
					if(pSubscription->nEventItemCount > 0 && pSubscription->pEventItems != 0)
					{
						if(nEventItemIndex < pSubscription->nEventItemCount)
						{
							BrbUaRcEventItemIntern_TYP* pEventItemInternOri = ((BrbUaRcEventItemIntern_TYP*)pSubscription->pEventItems) + nEventItemIndex;
							bResult = pEventItemInternOri->bEventReceived;
						}
					}
				}
			}
		}
	}
	return bResult;
}

// NOLINTEND(readability-*, bugprone-easily-swappable-parameters, bugprone-branch-clone, clang-diagnostic-invalid-utf8, clang-diagnostic-invalid-source-encoding, clang-diagnostic-pointer-arith, clang-diagnostic-strict-prototypes, hicpp-uppercase-literal-suffix, cppcoreguidelines-*, performance-*)
```

#### BrbUaRcGetEventItemReceiveCount.c
```c
#include <bur/plctypes.h>
#ifdef __cplusplus
	extern "C"
	{
#endif

#include "BrbLibUa.h"
#include <string.h>
#include <AnsiCFunc.h>

#ifdef __cplusplus
	};
#endif

// NOLINTBEGIN(readability-*, bugprone-easily-swappable-parameters, bugprone-branch-clone, clang-diagnostic-invalid-utf8, clang-diagnostic-invalid-source-encoding, clang-diagnostic-pointer-arith, clang-diagnostic-strict-prototypes, hicpp-uppercase-literal-suffix, cppcoreguidelines-*, performance-*)

/* Gibt zurück, ob ein Event empfangen wurde */
unsigned long BrbUaRcGetEventItemReceiveCount(struct BrbUaRunClient_TYP* pRunClient, unsigned short nSubscriptionIndex, unsigned short nEventItemIndex)
{
	UDINT nResult = 0;
	if(pRunClient != 0)
	{
		if(pRunClient->State.eClientState == eBRB_RCCLTSTATE_CONNECTED)
		{
			if(pRunClient->Subscriptions.nSubscriptionCount > 0 && pRunClient->Subscriptions.pSubscriptions != 0)
			{
				if(nSubscriptionIndex < pRunClient->Subscriptions.nSubscriptionCount)
				{
					BrbUaRcSubscriptionIntern_TYP* pSubscription = ((BrbUaRcSubscriptionIntern_TYP*)pRunClient->Subscriptions.pSubscriptions) + nSubscriptionIndex;
					if(pSubscription->nEventItemCount > 0 && pSubscription->pEventItems != 0)
					{
						if(nEventItemIndex < pSubscription->nEventItemCount)
						{
							BrbUaRcEventItemIntern_TYP* pEventItemInternOri = ((BrbUaRcEventItemIntern_TYP*)pSubscription->pEventItems) + nEventItemIndex;
							nResult = pEventItemInternOri->nReceiveCount;
						}
					}
				}
			}
		}
	}
	return nResult;
}

// NOLINTEND(readability-*, bugprone-easily-swappable-parameters, bugprone-branch-clone, clang-diagnostic-invalid-utf8, clang-diagnostic-invalid-source-encoding, clang-diagnostic-pointer-arith, clang-diagnostic-strict-prototypes, hicpp-uppercase-literal-suffix, cppcoreguidelines-*, performance-*)
```

#### BrbUaRcGetEventField.c
```c
#include <bur/plctypes.h>
#ifdef __cplusplus
	extern "C"
	{
#endif

#include "BrbLibUa.h"
#include <string.h>
#include <AnsiCFunc.h>

#ifdef __cplusplus
	};
#endif

// NOLINTBEGIN(readability-*, bugprone-easily-swappable-parameters, bugprone-branch-clone, clang-diagnostic-invalid-utf8, clang-diagnostic-invalid-source-encoding, clang-diagnostic-pointer-arith, clang-diagnostic-strict-prototypes, hicpp-uppercase-literal-suffix, cppcoreguidelines-*, performance-*)

/* Gibt ein ermitteltes EventField zurück */
unsigned short BrbUaRcGetEventField(struct BrbUaRunClient_TYP* pRunClient, unsigned short nSubscriptionIndex, unsigned short nEventItemIndex, unsigned short nEventFieldIndex, struct BrbUaRcEventField_TYP* pEventField)
{
	UINT nStatus = eBRB_ERR_NULL_POINTER;
	if(pRunClient != 0 && pEventField != 0)
	{
		memset(pEventField, 0, sizeof(BrbUaRcEventField_TYP));
		nStatus = eBRB_ERR_UA_NO_ELEMENTS;
		if(pRunClient->Subscriptions.nSubscriptionCount > 0 && pRunClient->Subscriptions.pSubscriptions != 0)
		{
			nStatus = eBRB_ERR_UA_INVALID_INDEX;
			if(nSubscriptionIndex < pRunClient->Subscriptions.nSubscriptionCount)
			{
				nStatus = eBRB_ERR_UA_NO_ELEMENTS;
				BrbUaRcSubscriptionIntern_TYP* pSubscription = ((BrbUaRcSubscriptionIntern_TYP*)pRunClient->Subscriptions.pSubscriptions) + nSubscriptionIndex;
				if(pSubscription->nEventItemCount > 0 && pSubscription->pEventItems != 0)
				{
					nStatus = eBRB_ERR_UA_INVALID_INDEX;
					if(nEventItemIndex < pSubscription->nEventItemCount)
					{
						nStatus = eBRB_ERR_UA_NO_ELEMENTS;
						BrbUaRcEventItemIntern_TYP* pEventItem = ((BrbUaRcEventItemIntern_TYP*)pSubscription->pEventItems) + nEventItemIndex;
						if(pEventItem->nEventFieldCount > 0 && pEventItem->pEfFieldSelections != 0 && pEventItem->pEfFieldVars != 0)
						{
							nStatus = eBRB_ERR_UA_INVALID_INDEX;
							if(nEventFieldIndex < pEventItem->nEventFieldCount)
							{
								nStatus = eBRB_ERR_OK;
								pEventField->nDatObjNamespaceIndex = *(((UINT*)pEventItem->pEfDatObjNamespaceIndices) + nEventFieldIndex);
								UARelativePath* pSelection = ((UARelativePath*)pEventItem->pEfFieldSelections) + nEventFieldIndex;
								memcpy(&pEventField->FieldSelection, pSelection, sizeof(UARelativePath));
								STRING sVarName[nBRBUA_VARNAME_TEXT_CHAR_MAX+1];
								STRING* pVar = (STRING*)((USINT*)pEventItem->pEfFieldVars) + (nEventFieldIndex * sizeof(sVarName));
								BrbStringCopy(pEventField->sVar, pVar, sizeof(pEventField->sVar));
							}
						}
					}
				}
			}
		}
	}
	return nStatus;
}

// NOLINTEND(readability-*, bugprone-easily-swappable-parameters, bugprone-branch-clone, clang-diagnostic-invalid-utf8, clang-diagnostic-invalid-source-encoding, clang-diagnostic-pointer-arith, clang-diagnostic-strict-prototypes, hicpp-uppercase-literal-suffix, cppcoreguidelines-*, performance-*)
```

#### BrbUaRcMonitor.c
```c
#include <bur/plctypes.h>
#ifdef __cplusplus
	extern "C"
	{
#endif

#include "BrbLibUa.h"
#include <string.h>
#include <AnsiCFunc.h>

#ifdef __cplusplus
	};
#endif

// NOLINTBEGIN(readability-*, bugprone-easily-swappable-parameters, bugprone-branch-clone, clang-diagnostic-invalid-utf8, clang-diagnostic-invalid-source-encoding, clang-diagnostic-pointer-arith, clang-diagnostic-strict-prototypes, hicpp-uppercase-literal-suffix, cppcoreguidelines-*, performance-*)

/* Zeigt die Inhalte des internen Speichers */
unsigned short BrbUaRcMonitor(struct BrbUaRunClient_TYP* pRunClient, struct BrbUaRcMonitor_TYP* pMonitor)
{
	UINT nStatus = eBRB_ERR_NULL_POINTER;
	if(pRunClient != 0 && pMonitor != 0)
	{
		nStatus = eBRB_ERR_NOT_ENABLED;
		if(pMonitor->bEnable == 1)
		{
			nStatus = eBRB_ERR_OK;
			brsmemset((UDINT)&pMonitor->Namespace.Namespace , 0, sizeof(pMonitor->Namespace.Namespace));
			BrbUaRcGetSrvNamespace(pRunClient, pMonitor->Namespace.nDatObjNamespaceIndex, &pMonitor->Namespace.Namespace);

			brsmemset((UDINT)&pMonitor->NodeHandle.NodeHandle , 0, sizeof(pMonitor->NodeHandle.NodeHandle));
			pMonitor->NodeHandle.nMonitorStatus = BrbUaRcGetNodeHandle(pRunClient, pMonitor->NodeHandle.nNodeHandleIndex, &pMonitor->NodeHandle.NodeHandle);

			brsmemset((UDINT)&pMonitor->ReadBlock.ReadBlock, 0, sizeof(pMonitor->ReadBlock.ReadBlock));
			brsmemset((UDINT)&pMonitor->ReadBlock.ReadBlockIntern, 0, sizeof(pMonitor->ReadBlock.ReadBlockIntern));
			pMonitor->ReadBlock.nMonitorStatus = BrbUaRcGetReadBlock(pRunClient, pMonitor->ReadBlock.nReadBlockIndex, &pMonitor->ReadBlock.ReadBlock, &pMonitor->ReadBlock.ReadBlockIntern);

			brsmemset((UDINT)&pMonitor->ReadItem.ReadItem, 0, sizeof(pMonitor->ReadItem.ReadItem));
			pMonitor->ReadItem.nMonitorStatus = BrbUaRcGetReadItem(pRunClient, pMonitor->ReadItem.nReadBlockIndex, pMonitor->ReadItem.nReadItemIndex, &pMonitor->ReadItem.ReadItem);

			brsmemset((UDINT)&pMonitor->WriteBlock.WriteBlock, 0, sizeof(pMonitor->WriteBlock.WriteBlock));
			brsmemset((UDINT)&pMonitor->WriteBlock.WriteBlockIntern, 0, sizeof(pMonitor->WriteBlock.WriteBlockIntern));
			pMonitor->WriteBlock.nMonitorStatus = BrbUaRcGetWriteBlock(pRunClient, pMonitor->WriteBlock.nWriteBlockIndex, &pMonitor->WriteBlock.WriteBlock, &pMonitor->WriteBlock.WriteBlockIntern);

			brsmemset((UDINT)&pMonitor->WriteItem.WriteItem, 0, sizeof(pMonitor->WriteItem.WriteItem));
			pMonitor->WriteItem.nMonitorStatus = BrbUaRcGetWriteItem(pRunClient, pMonitor->WriteItem.nWriteBlockIndex, pMonitor->WriteItem.nWriteItemIndex, &pMonitor->WriteItem.WriteItem);

			brsmemset((UDINT)&pMonitor->Method.Method, 0, sizeof(pMonitor->Method.Method));
			pMonitor->Method.nMonitorStatus = BrbUaRcGetMethod(pRunClient, pMonitor->Method.nMethodIndex, &pMonitor->Method.Method, & pMonitor->Method.MethodIntern);

			brsmemset((UDINT)&pMonitor->Argument.Argument, 0, sizeof(pMonitor->Argument.Argument));
			pMonitor->Argument.nMonitorStatus = BrbUaRcGetArgument(pRunClient, pMonitor->Argument.nMethodIndex, pMonitor->Argument.bOutput, pMonitor->Argument.nArgumentIndex, &pMonitor->Argument.Argument);

			brsmemset((UDINT)&pMonitor->Subscription.Subscription, 0, sizeof(pMonitor->Subscription.Subscription));
			brsmemset((UDINT)&pMonitor->Subscription.SubscriptionIntern, 0, sizeof(pMonitor->Subscription.SubscriptionIntern));
			pMonitor->Subscription.nMonitorStatus = BrbUaRcGetSubscription(pRunClient, pMonitor->Subscription.nSubscriptionIndex, &pMonitor->Subscription.Subscription, &pMonitor->Subscription.SubscriptionIntern);

			brsmemset((UDINT)&pMonitor->MonitoredItem.MonitoredItem, 0, sizeof(pMonitor->MonitoredItem.MonitoredItem));
			pMonitor->MonitoredItem.nMonitorStatus = BrbUaRcGetMonitoredItem(pRunClient, pMonitor->MonitoredItem.nSubscriptionIndex, pMonitor->MonitoredItem.nMonitoredItemIndex, &pMonitor->MonitoredItem.MonitoredItem);

			brsmemset((UDINT)&pMonitor->EventItem.EventItem, 0, sizeof(pMonitor->EventItem.EventItem));
			brsmemset((UDINT)&pMonitor->EventItem.EventItemIntern, 0, sizeof(pMonitor->EventItem.EventItemIntern));
			pMonitor->EventItem.nMonitorStatus = BrbUaRcGetEventItem(pRunClient, pMonitor->EventItem.nSubscriptionIndex, pMonitor->EventItem.nEventItemIndex, &pMonitor->EventItem.EventItem, &pMonitor->EventItem.EventItemIntern);

			brsmemset((UDINT)&pMonitor->EventField.EventField, 0, sizeof(pMonitor->EventField.EventField));
			pMonitor->EventField.nMonitorStatus = BrbUaRcGetEventField(pRunClient, pMonitor->EventField.nSubscriptionIndex, pMonitor->EventField.nEventItemIndex, pMonitor->EventField.nEventFieldIndex, &pMonitor->EventField.EventField);
		}
		else
		{
			brsmemset((UDINT)&pMonitor->Namespace.Namespace , 0, sizeof(pMonitor->Namespace.Namespace));
			pMonitor->NodeHandle.nMonitorStatus = eBRB_ERR_NOT_ENABLED;
			brsmemset((UDINT)&pMonitor->NodeHandle.NodeHandle , 0, sizeof(pMonitor->NodeHandle.NodeHandle));
			pMonitor->ReadBlock.nMonitorStatus = eBRB_ERR_NOT_ENABLED;
			brsmemset((UDINT)&pMonitor->ReadBlock.ReadBlock, 0, sizeof(pMonitor->ReadBlock.ReadBlock));
			brsmemset((UDINT)&pMonitor->ReadBlock.ReadBlockIntern, 0, sizeof(pMonitor->ReadBlock.ReadBlockIntern));
			pMonitor->ReadItem.nMonitorStatus = eBRB_ERR_NOT_ENABLED;
			brsmemset((UDINT)&pMonitor->ReadItem.ReadItem, 0, sizeof(pMonitor->ReadItem.ReadItem));
			pMonitor->WriteBlock.nMonitorStatus = eBRB_ERR_NOT_ENABLED;
			brsmemset((UDINT)&pMonitor->WriteBlock.WriteBlock, 0, sizeof(pMonitor->WriteBlock.WriteBlock));
			brsmemset((UDINT)&pMonitor->WriteBlock.WriteBlockIntern, 0, sizeof(pMonitor->WriteBlock.WriteBlockIntern));
			pMonitor->WriteItem.nMonitorStatus = eBRB_ERR_NOT_ENABLED;
			brsmemset((UDINT)&pMonitor->WriteItem.WriteItem, 0, sizeof(pMonitor->WriteItem.WriteItem));
			pMonitor->Method.nMonitorStatus = eBRB_ERR_NOT_ENABLED;
			brsmemset((UDINT)&pMonitor->Method.Method, 0, sizeof(pMonitor->Method.Method));
			pMonitor->Argument.nMonitorStatus = eBRB_ERR_NOT_ENABLED;
			brsmemset((UDINT)&pMonitor->Argument.Argument, 0, sizeof(pMonitor->Argument.Argument));
			pMonitor->Subscription.nMonitorStatus = eBRB_ERR_NOT_ENABLED;
			brsmemset((UDINT)&pMonitor->Subscription.Subscription, 0, sizeof(pMonitor->Subscription.Subscription));
			brsmemset((UDINT)&pMonitor->Subscription.SubscriptionIntern, 0, sizeof(pMonitor->Subscription.SubscriptionIntern));
			pMonitor->MonitoredItem.nMonitorStatus = eBRB_ERR_NOT_ENABLED;
			brsmemset((UDINT)&pMonitor->MonitoredItem.MonitoredItem, 0, sizeof(pMonitor->MonitoredItem.MonitoredItem));
			pMonitor->EventItem.nMonitorStatus = eBRB_ERR_NOT_ENABLED;
			brsmemset((UDINT)&pMonitor->EventItem.EventItem, 0, sizeof(pMonitor->EventItem.EventItem));
			brsmemset((UDINT)&pMonitor->EventItem.EventItemIntern, 0, sizeof(pMonitor->EventItem.EventItemIntern));
			pMonitor->EventField.nMonitorStatus = eBRB_ERR_NOT_ENABLED;
			brsmemset((UDINT)&pMonitor->EventField.EventField, 0, sizeof(pMonitor->EventField.EventField));
		}
		pMonitor->nMonitorStatus = nStatus;
	}
	return nStatus;
}

// NOLINTEND(readability-*, bugprone-easily-swappable-parameters, bugprone-branch-clone, clang-diagnostic-invalid-utf8, clang-diagnostic-invalid-source-encoding, clang-diagnostic-pointer-arith, clang-diagnostic-strict-prototypes, hicpp-uppercase-literal-suffix, cppcoreguidelines-*, performance-*)
```

#### Package Logical/Libraries/BrbLibUa/Server/Methods - Funktionen für OpcUa-Methoden

#### BrbUaSrvHandleMethod.c - Behandelt einen Methoden-Aufruf
```c
#include <bur/plctypes.h>
#ifdef __cplusplus
	extern "C"
	{
#endif

#include "BrbLibUa.h"
#include <AnsiCFunc.h>
#include <string.h>

#ifdef __cplusplus
	};
#endif

// NOLINTBEGIN(readability-*, bugprone-easily-swappable-parameters, bugprone-branch-clone, clang-diagnostic-invalid-utf8, clang-diagnostic-invalid-source-encoding, clang-diagnostic-pointer-arith, clang-diagnostic-strict-prototypes, hicpp-uppercase-literal-suffix, cppcoreguidelines-*, performance-*)

/* Behandelt einen Methoden-Aufruf */
plcdword BrbUaSrvHandleMethod(struct BrbUaSrvMethod_TYP* pMethod)
{
	DWORD nStatus = 0x80460000; // = Bad_StructureMissing
	if(pMethod != 0)
	{
		nStatus = 0x00000000; // = Good
		if(pMethod->Par.bEnable == 1)
		{
			pMethod->Intern.bEnabled = 1;
		}
		if(pMethod->Intern.bEnabled == 1)
		{
			switch(pMethod->Intern.nStep)
			{
				case 0: // Init
					BrbStringCopy(pMethod->Intern.fbUaSrv_MethodOperate.MethodName, pMethod->Par.sMethodName, sizeof(pMethod->Intern.fbUaSrv_MethodOperate.MethodName));
					pMethod->Intern.nErrorId = 0;
					pMethod->Intern.fbUaSrv_MethodOperate.Action = UaMoa_CheckIsCalled;	// Abfrage über Baustein
					pMethod->Intern.fbUaSrv_MethodOperate.Execute = 1;
					pMethod->Intern.nStep = 1;
					break;

				case 1: // Prüfen, ob Methode aufgerufen ist
					UaSrv_MethodOperate(&pMethod->Intern.fbUaSrv_MethodOperate);
					if(pMethod->Intern.fbUaSrv_MethodOperate.Busy == 0)
					{
						if(pMethod->Intern.fbUaSrv_MethodOperate.Done == 1)
						{
							if(pMethod->Intern.fbUaSrv_MethodOperate.IsCalled == 1)
							{
								// Methode ist aufgerufen -> Ausführung
								pMethod->State.bExecuteUserCode = 1;
								pMethod->State.bExecuteUserCodeInit = 1;
								pMethod->Par.bUserCodeIsFinished = 0;
								pMethod->State.nCallCount += 1;
								pMethod->Intern.fbUaSrv_MethodOperate.Execute = 0;
								UaSrv_MethodOperate(&pMethod->Intern.fbUaSrv_MethodOperate);
								pMethod->Intern.nStep = 2;
							}
							else if(pMethod->Par.bEnable == 0)
							{
								// Ausführung soll und kann beendet werden
								pMethod->Intern.fbUaSrv_MethodOperate.Execute = 0;
								UaSrv_MethodOperate(&pMethod->Intern.fbUaSrv_MethodOperate);
								pMethod->Intern.bEnabled = 0;
								pMethod->Intern.nStep = 0;
							}
							else
							{
								// Weiter prüfen
								pMethod->Intern.fbUaSrv_MethodOperate.Execute = 0;
								UaSrv_MethodOperate(&pMethod->Intern.fbUaSrv_MethodOperate);
								pMethod->Intern.fbUaSrv_MethodOperate.Execute = 1;
							}
						}
						else if(pMethod->Intern.fbUaSrv_MethodOperate.Error == 1)
						{
							// Fehler
							pMethod->Intern.nErrorId = pMethod->Intern.fbUaSrv_MethodOperate.ErrorID;
							pMethod->State.nLastErrorId = pMethod->Intern.fbUaSrv_MethodOperate.ErrorID;
							pMethod->State.eLastErrorAction = pMethod->Intern.fbUaSrv_MethodOperate.Action;
							pMethod->State.nErrorCount += 1;
							pMethod->Intern.fbUaSrv_MethodOperate.Execute = 0;
							UaSrv_MethodOperate(&pMethod->Intern.fbUaSrv_MethodOperate);
							pMethod->Intern.nStep = 4;
						}
					}
					break;

				case 2:	// Warten auf Ausführung des User-Codes
					pMethod->State.bExecuteUserCodeInit = 0;
					if(pMethod->Par.bUserCodeIsFinished == 1)
					{
						// User-Code ist fertig ausgeführt
						pMethod->State.bExecuteUserCode = 0;
						pMethod->Par.bUserCodeIsFinished = 0;
						BrbStringCopy(pMethod->Intern.fbUaSrv_MethodOperate.MethodName, pMethod->Par.sMethodName, sizeof(pMethod->Intern.fbUaSrv_MethodOperate.MethodName));
						pMethod->Intern.fbUaSrv_MethodOperate.Action = UaMoa_Finished;	// Rückmeldung an Baustein
						pMethod->Intern.fbUaSrv_MethodOperate.Execute = 1;
						pMethod->Intern.nStep = 3;
					}
					break;

				case 3:	// Ausführung rückmelden
					UaSrv_MethodOperate(&pMethod->Intern.fbUaSrv_MethodOperate);
					if(pMethod->Intern.fbUaSrv_MethodOperate.Busy == 0)
					{
						if(pMethod->Intern.fbUaSrv_MethodOperate.Done == 1)
						{
							// Bereit für neuen Aufruf
							if(pMethod->Par.bEnable == 0)
							{
								// Ausführung soll und kann beendet werden
								pMethod->Intern.bEnabled = 0;
							}
							pMethod->Intern.fbUaSrv_MethodOperate.Execute = 0;
							UaSrv_MethodOperate(&pMethod->Intern.fbUaSrv_MethodOperate);
							pMethod->Intern.nStep = 0;
						}
						else if(pMethod->Intern.fbUaSrv_MethodOperate.Error == 1)
						{
							// Fehler
							pMethod->Intern.nErrorId = pMethod->Intern.fbUaSrv_MethodOperate.ErrorID;
							pMethod->State.nLastErrorId = pMethod->Intern.fbUaSrv_MethodOperate.ErrorID;
							pMethod->State.eLastErrorAction = pMethod->Intern.fbUaSrv_MethodOperate.Action;
							pMethod->State.nErrorCount += 1;
							pMethod->Intern.fbUaSrv_MethodOperate.Execute = 0;
							UaSrv_MethodOperate(&pMethod->Intern.fbUaSrv_MethodOperate);
							pMethod->Intern.nStep = 4;
						}
					}
					break;

				case 4:	// Fehler im Baustein
					nStatus = pMethod->Intern.nErrorId;
					pMethod->State.bExecuteUserCode = 0;
					pMethod->Par.bUserCodeIsFinished = 0;
					pMethod->Intern.fbUaSrv_MethodOperate.Execute = 0;
					UaSrv_MethodOperate(&pMethod->Intern.fbUaSrv_MethodOperate);
					if(pMethod->Par.bEnable == 0)
					{
						// Ausführung soll und kann beendet werden
						pMethod->Intern.bEnabled = 0;
					}
					pMethod->Intern.nStep = 0;
					break;

			}
			BrbUaGetStatusCodeText(pMethod->State.nLastErrorId, pMethod->State.sLastErrorId, sizeof(pMethod->State.sLastErrorId));
		}
	}
	return nStatus;
}

// NOLINTEND(readability-*, bugprone-easily-swappable-parameters, bugprone-branch-clone, clang-diagnostic-invalid-utf8, clang-diagnostic-invalid-source-encoding, clang-diagnostic-pointer-arith, clang-diagnostic-strict-prototypes, hicpp-uppercase-literal-suffix, cppcoreguidelines-*, performance-*)
```

#### BrbUaSrvGetMethodOperateText.c
```c
#include <bur/plctypes.h>
#ifdef __cplusplus
	extern "C"
	{
#endif

#include "BrbLibUa.h"
#include <string.h>

#ifdef __cplusplus
	};
#endif

// NOLINTBEGIN(readability-*, bugprone-easily-swappable-parameters, bugprone-branch-clone, clang-diagnostic-invalid-utf8, clang-diagnostic-invalid-source-encoding, clang-diagnostic-pointer-arith, clang-diagnostic-strict-prototypes, hicpp-uppercase-literal-suffix, cppcoreguidelines-*, performance-*)

/* Gibt den Text einer MethodOperateAction zurück */
plcdword BrbUaSrvGetMethodOperateText(enum UaMethodOperateAction eAction, plcstring* pActionText, unsigned long nActionTextSize)
{
	DWORD nStatus = 0x80460000; // = Bad_StructureMissing
	if(pActionText != 0)
	{
		nStatus = 0x00000000; // = Good
		memset(pActionText, 0, nActionTextSize);
		switch(eAction) // NOLINT(hicpp-multiway-paths-covered)
		{
			case UaMoa_CheckIsCalled:
				BrbStringCat(pActionText, "CheckIsCalled", nActionTextSize);
				break;

			case UaMoa_Finished:
				BrbStringCat(pActionText, "Finished", nActionTextSize);
				break;

		}
	}
	return nStatus;
}

// NOLINTEND(readability-*, bugprone-easily-swappable-parameters, bugprone-branch-clone, clang-diagnostic-invalid-utf8, clang-diagnostic-invalid-source-encoding, clang-diagnostic-pointer-arith, clang-diagnostic-strict-prototypes, hicpp-uppercase-literal-suffix, cppcoreguidelines-*, performance-*)
```

#### BrbUaRunServerInit.c
```c
#include <bur/plctypes.h>
#ifdef __cplusplus
	extern "C"
	{
#endif

#include "BrbLibUa.h"
#include <string.h>
#include <AnsiCFunc.h>

#ifdef __cplusplus
	};
#endif

// NOLINTBEGIN(readability-*, bugprone-easily-swappable-parameters, bugprone-branch-clone, clang-diagnostic-invalid-utf8, clang-diagnostic-invalid-source-encoding, clang-diagnostic-pointer-arith, clang-diagnostic-strict-prototypes, hicpp-uppercase-literal-suffix, cppcoreguidelines-*, performance-*)

// Prototypen
BOOL ParseServerValue(STRING** ppStart, STRING* pPar, STRING* pValue);

// Eigene Enums und Typen
enum Steps_ENUM
{
	eSTEP_INIT,
	eSTEP_GET_DAT_INFO,
	eSTEP_COUNT_GENERAL,
	eSTEP_ALLOC_NAMESPACES,
	eSTEP_ALLOC_EVENTS,
	eSTEP_PARSE_GENERAL,
	eSTEP_ALLOC_EVENT_FIELDS,
	eSTEP_PARSE_EVENT_FIELDS,
	eSTEP_FINISHED,
};

/* Initialisiert eine Client-Instanz */
void BrbUaRunServerInit(struct BrbUaRunServerInit* inst)
{
	switch(inst->eStep)
	{
		case eSTEP_INIT:
			// Fub initialisieren
			inst->nStatus =  eBRB_ERR_BUSY;
			memset(&inst->fbDatObjInfo, 0, sizeof(inst->fbDatObjInfo));
			memset(&inst->fbDatObjRead, 0, sizeof(inst->fbDatObjRead));
			// Client-Pointer prüfen
			if(inst->pRunServer != 0)
			{
				inst->pRunServer->State.eState = eBRB_RSSTATE_INITIALIZING;
				inst->pRunServer->State.nErroId = 0x00000000;
				strcpy(inst->pRunServer->State.sErrorText, "");
				inst->pRunServer->State.eServerState = UASS_Shutdown;
				memset(&inst->pRunServer->Namespaces, 0, sizeof(inst->pRunServer->Namespaces));
				memset(&inst->pRunServer->Events, 0, sizeof(inst->pRunServer->Events));
				inst->pRunServer->Events.nEventCount = 0;
				inst->pRunServer->Events.nFieldsCountTotal = 0;
				inst->eStep = eSTEP_GET_DAT_INFO;
			}
			else
			{
				inst->nStatus = eBRB_ERR_NULL_POINTER;
				inst->eStep = eSTEP_INIT;
			}
			break;

		case eSTEP_GET_DAT_INFO:
			// Datenobjekt-Ident ermitteln
			inst->nStatus  = eBRB_ERR_BUSY;
			inst->fbDatObjInfo.enable = 1;
			inst->fbDatObjInfo.pName = (UDINT)&inst->pRunServer->Cfg.sCfgDataObjName;
			DatObjInfo(&inst->fbDatObjInfo);
			if(inst->fbDatObjInfo.status == 0)
			{
				inst->eStep = eSTEP_COUNT_GENERAL;
			}
			else if(inst->fbDatObjInfo.status != eBRB_ERR_BUSY)
			{
				// Fehler
				inst->nStatus = inst->fbDatObjInfo.status;
				inst->pRunServer->State.nErroId = inst->nStatus;
				strcpy(inst->pRunServer->State.sErrorText, "Init error on getting data object info");
				inst->pRunServer->State.eState = eBRB_RSSTATE_INIT_ERROR;
				inst->eStep = eSTEP_INIT;
			}
			break;

		case eSTEP_COUNT_GENERAL:
			// Elemente in Datenobjekt zählen
			inst->nStatus  = eBRB_ERR_BUSY;
			inst->pRunServer->Namespaces.nNamespaceCount = (UINT)BrbStringCountText((STRING*)inst->fbDatObjInfo.pDatObjMem, nBRBUA_KEYWORD_NAMESPACE, inst->fbDatObjInfo.len);
			inst->nNamespaceIndex = -1;
			inst->pRunServer->Events.nEventCount = (UINT)BrbStringCountText((STRING*)inst->fbDatObjInfo.pDatObjMem, nBRBUA_KEYWORD_EVENT, inst->fbDatObjInfo.len);
			inst->pRunServer->Events.nFieldsCountTotal = BrbStringCountText((STRING*)inst->fbDatObjInfo.pDatObjMem, nBRBUA_KEYWORD_EVENT_FIELD, inst->fbDatObjInfo.len);
			inst->nEventIndex = -1;
			inst->nEventFieldIndex = 0;
			inst->eStep = eSTEP_ALLOC_NAMESPACES;
			break;

		case eSTEP_ALLOC_NAMESPACES:
			// Speicher für Namespaces allokieren
			inst->nStatus  = eBRB_ERR_BUSY;
			if(inst->pRunServer->Namespaces.nNamespaceCount > 0)
			{
				inst->pRunServer->Namespaces.nMemLen = inst->pRunServer->Namespaces.nNamespaceCount * sizeof(BrbUaRsNamespace_TYP);
				inst->nAllocStatus = TMP_alloc(inst->pRunServer->Namespaces.nMemLen, (void*)&inst->pRunServer->Namespaces.pNamespaces);
				if(inst->nAllocStatus == 0 && inst->pRunServer->Namespaces.pNamespaces != 0)
				{
					memset((USINT*)inst->pRunServer->Namespaces.pNamespaces, 0, inst->pRunServer->Namespaces.nMemLen);
					inst->eStep = eSTEP_ALLOC_EVENTS;
				}
				else
				{
					// Fehler
					inst->nStatus = inst->nAllocStatus;
					inst->pRunServer->State.nErroId = inst->nStatus;
					strcpy(inst->pRunServer->State.sErrorText, "Init error on allocating memory for namespaces");
					inst->pRunServer->State.eState = eBRB_RSSTATE_INIT_ERROR;
					inst->eStep = eSTEP_INIT;
				}
			}
			else
			{
				// Keine Namespaces angegeben
				inst->eStep = eSTEP_ALLOC_EVENTS;
			}
			break;

		case eSTEP_ALLOC_EVENTS:
			// Speicher für Events allokieren
			inst->nStatus  = eBRB_ERR_BUSY;
			if(inst->pRunServer->Events.nEventCount > 0)
			{
				inst->pRunServer->Events.nMemLen = inst->pRunServer->Events.nEventCount * sizeof(BrbUaRsEventIntern_TYP);
				inst->nAllocStatus = TMP_alloc(inst->pRunServer->Events.nMemLen, (void*)&inst->pRunServer->Events.pEvents);
				if(inst->nAllocStatus == 0 && inst->pRunServer->Events.pEvents != 0)
				{
					memset((USINT*)inst->pRunServer->Events.pEvents, 0, inst->pRunServer->Events.nMemLen);
					inst->eStep = eSTEP_PARSE_GENERAL;
				}
				else
				{
					// Fehler
					inst->nStatus = inst->nAllocStatus;
					inst->pRunServer->State.nErroId = inst->nStatus;
					strcpy(inst->pRunServer->State.sErrorText, "Init error on allocating memory for events");
					inst->pRunServer->State.eState = eBRB_RSSTATE_INIT_ERROR;
					inst->eStep = eSTEP_INIT;
					break;
				}
			}
			else
			{
				// Keine Subscriptions angegeben
				inst->eStep = eSTEP_PARSE_GENERAL;
			}
			break;

		case eSTEP_PARSE_GENERAL:
			// Datenobjekt parsen
			inst->nStatus  = eBRB_ERR_BUSY;
			for(inst->nLoopIndex=0; inst->nLoopIndex<nBRBUA_SRV_READ_LINES; inst->nLoopIndex++) // In einem Zyklus 100 Zeilen lesen
			{
				inst->fbDatObjRead.enable = 1;
				inst->fbDatObjRead.ident = inst->fbDatObjInfo.ident;
				inst->fbDatObjRead.pDestination = (UDINT)&inst->sLine;
				inst->fbDatObjRead.len = sizeof(inst->sLine)-1;
				if(inst->fbDatObjInfo.len < inst->fbDatObjRead.Offset + inst->fbDatObjRead.len)
				{
					// Es können nur mehr eine bestimmte Anzahl von Bytes gelesen werden
					inst->fbDatObjRead.len = inst->fbDatObjInfo.len - inst->fbDatObjRead.Offset;
				}
				DatObjRead(&inst->fbDatObjRead);
				if(inst->fbDatObjRead.status == 0)
				{
					inst->nLineLen = strlen(inst->sLine);
					if(BrbStringStartsWith(inst->sLine, nBRBUA_KEYWORD_NAMESPACE) == 1)
					{
						inst->nNamespaceIndex++;
						if(inst->nNamespaceIndex < inst->pRunServer->Namespaces.nNamespaceCount && inst->pRunServer->Namespaces.pNamespaces != 0)
						{
							// Werte des Namespaces auslesen
							BrbUaRsNamespace_TYP* pNamespace = ((BrbUaRsNamespace_TYP*)inst->pRunServer->Namespaces.pNamespaces) + inst->nNamespaceIndex;
							STRING* pStart = (STRING*)&inst->sLine;
							memset(&inst->sValue, 0, sizeof(inst->sValue));
							if(ParseServerValue(&pStart, "Uri=", inst->sValue) == 1)
							{
								BrbStringCopy(pNamespace->sNamespaceUri, inst->sValue, sizeof(pNamespace->sNamespaceUri));
							}
						}
					}
					else if(BrbStringStartsWith(inst->sLine, nBRBUA_KEYWORD_EVENT) == 1)
					{
						inst->nEventIndex++;
						if(inst->nEventIndex < inst->pRunServer->Events.nEventCount && inst->pRunServer->Events.pEvents != 0)
						{
							BrbUaRsEventIntern_TYP* pEvent = ((BrbUaRsEventIntern_TYP*)inst->pRunServer->Events.pEvents) + inst->nEventIndex;
							// Zuerst Default-Werte setzen
							pEvent->nDatObjNamespaceIndex = 0;
							BrbUaSetNodeId(&pEvent->TypeNodeId, "2041", 0);// Server-NamespaceIndex muss erst noch ermittelt werden
							// Werte des Events auslesen
							STRING* pStart = (STRING*)&inst->sLine;
							memset(&inst->sValue, 0, sizeof(inst->sValue));
							if(ParseServerValue(&pStart, "TypeNs=", inst->sValue) == 1)
							{
								inst->nValue = brsatoi((UDINT)&inst->sValue);
								pEvent->nDatObjNamespaceIndex = (UINT)inst->nValue;
							}
							if(ParseServerValue(&pStart, "TypeId=", inst->sValue) == 1)
							{
								BrbUaSetNodeId(&pEvent->TypeNodeId, inst->sValue, 0);// Server-NamespaceIndex muss erst noch ermittelt werden
							}
						}
					}
					else if(BrbStringStartsWith(inst->sLine, nBRBUA_KEYWORD_EVENT_FIELD) == 1)
					{
						// Fields zählen
						if(inst->nEventIndex < inst->pRunServer->Events.nEventCount && inst->pRunServer->Events.pEvents != 0)
						{
							BrbUaRsEventIntern_TYP* pEvent = ((BrbUaRsEventIntern_TYP*)inst->pRunServer->Events.pEvents) + inst->nEventIndex;
							pEvent->nFieldCount++;
						}
					}
					// Nächste Zeile lesen
					inst->fbDatObjRead.Offset += inst->nLineLen+1;
				}
				else if(inst->fbDatObjRead.status == doERR_ILLEGALLENGTH)
				{
					// Am Ende des Datenobjekts angelangt
					inst->fbDatObjRead.Offset = 0;
					inst->nEventIndex = 0;
					inst->eStep = eSTEP_ALLOC_EVENT_FIELDS;
					break;
				}
				else if(inst->fbDatObjRead.status != 65535)
				{
					// Fehler
					inst->nStatus = inst->fbDatObjRead.status;
					inst->pRunServer->State.nErroId = inst->nStatus;
					strcpy(inst->pRunServer->State.sErrorText, "Init error on parsing data object for general data");
					inst->pRunServer->State.eState = eBRB_RSSTATE_INIT_ERROR;
					inst->eStep = eSTEP_INIT;
					break;
				}
			}
			break;

		case eSTEP_ALLOC_EVENT_FIELDS:
			// Speicher für Fields pro Event allokieren
			inst->nStatus  = eBRB_ERR_BUSY;
			if(inst->pRunServer->Events.nEventCount > 0 && inst->pRunServer->Events.pEvents != 0)
			{
				if(inst->nEventIndex < inst->pRunServer->Events.nEventCount)
				{
					BrbUaRsEventIntern_TYP* pEvent = (((BrbUaRsEventIntern_TYP*)inst->pRunServer->Events.pEvents)  + inst->nEventIndex);
					if(pEvent->nFieldCount > 0)
					{
						pEvent->nMemLen = pEvent->nFieldCount * sizeof(UaSrv_FireEventFieldType);
						inst->nAllocStatus = TMP_alloc(pEvent->nMemLen, (void*)&pEvent->pFields);
						if(inst->nAllocStatus == 0 && pEvent->pFields != 0)
						{
							memset((USINT*)pEvent->pFields, 0, pEvent->nMemLen);
							inst->nEventIndex++;
						}
						else
						{
							// Fehler
							inst->nStatus = inst->nAllocStatus;
							inst->pRunServer->State.nErroId = inst->nStatus;
							BrbStringCopy(inst->pRunServer->State.sErrorText, "Init error on allocating memory for Fields of Event", sizeof(inst->pRunServer->State.sErrorText));
							STRING sHelp[16];
							brsitoa(inst->nEventIndex, (UDINT)&sHelp);
							BrbStringCat(inst->pRunServer->State.sErrorText, sHelp, sizeof(inst->pRunServer->State.sErrorText));
							inst->pRunServer->State.eState = eBRB_RSSTATE_INIT_ERROR;
							inst->eStep = eSTEP_INIT;
							break;
						}
					}
					else
					{
						inst->nEventIndex++;
					}
				}
				else
				{
					inst->nEventIndex = -1;
					inst->nEventFieldIndex = 0;
					inst->eStep = eSTEP_PARSE_EVENT_FIELDS;
				}
			}
			else
			{
				// Keine Events angegeben
				inst->eStep = eSTEP_FINISHED;
			}
			break;

		case eSTEP_PARSE_EVENT_FIELDS:
			// Parameter der Fields parsen
			inst->nStatus  = eBRB_ERR_BUSY;
			for(inst->nLoopIndex=0; inst->nLoopIndex<nBRBUA_SRV_READ_LINES; inst->nLoopIndex++) // In einem Zyklus 100 Zeilen lesen
			{
				inst->fbDatObjRead.enable = 1;
				inst->fbDatObjRead.ident = inst->fbDatObjInfo.ident;
				inst->fbDatObjRead.pDestination = (UDINT)&inst->sLine;
				inst->fbDatObjRead.len = sizeof(inst->sLine)-1;
				if(inst->fbDatObjInfo.len < inst->fbDatObjRead.Offset + inst->fbDatObjRead.len)
				{
					// Es können nur mehr eine bestimmte Anzahl von Bytes gelesen werden
					inst->fbDatObjRead.len = inst->fbDatObjInfo.len - inst->fbDatObjRead.Offset;
				}
				DatObjRead(&inst->fbDatObjRead);
				if(inst->fbDatObjRead.status == 0)
				{
					inst->nLineLen = strlen(inst->sLine);
					if(BrbStringStartsWith(inst->sLine, nBRBUA_KEYWORD_EVENT) == 1)
					{
						inst->nEventIndex++;
						inst->nEventFieldIndex = 0;
					}
					else if(BrbStringStartsWith(inst->sLine, nBRBUA_KEYWORD_EVENT_FIELD) == 1)
					{
						// Werte des Fields auslesen
						if(inst->nEventIndex < inst->pRunServer->Events.nEventCount && inst->pRunServer->Events.pEvents != 0)
						{
							BrbUaRsEventIntern_TYP* pEvent = ((BrbUaRsEventIntern_TYP*)inst->pRunServer->Events.pEvents) + inst->nEventIndex;
							if(inst->nEventFieldIndex < pEvent->nFieldCount)
							{
								UaSrv_FireEventFieldType* pEventField = ((UaSrv_FireEventFieldType*)pEvent->pFields) + inst->nEventFieldIndex;
								// Zuerst Default-Werte setzen
								pEventField->ErrorID = 0;
								// Dann exisitierende Parameter auslesen
								STRING* pStart = (STRING*)&inst->sLine;
								memset(&inst->sValue, 0, sizeof(inst->sValue));
								if(ParseServerValue(&pStart, "Name=", inst->sValue) == 1)
								{
									BrbStringCopy(pEventField->BrowsePath, inst->sValue, sizeof(pEventField->BrowsePath));
								}
								if(ParseServerValue(&pStart, "Var=", inst->sValue) == 1)
								{
									BrbStringCopy(pEventField->Variable, inst->sValue, sizeof(pEventField->Variable));
								}
							}
							inst->nEventFieldIndex++;
						}
					}
					// Nächste Zeile lesen
					inst->fbDatObjRead.Offset += inst->nLineLen+1;
				}
				else if(inst->fbDatObjRead.status == doERR_ILLEGALLENGTH)
				{
					// Am Ende des Datenobjekts angelangt
					inst->fbDatObjRead.Offset = 0;
					inst->nEventIndex = -1;
					inst->nEventFieldIndex = -1;
					inst->eStep = eSTEP_FINISHED;
					break;
				}
				else if(inst->fbDatObjRead.status != 65535)
				{
					// Fehler
					inst->nStatus = inst->fbDatObjRead.status;
					inst->pRunServer->State.nErroId = inst->nStatus;
					strcpy(inst->pRunServer->State.sErrorText, "Init error on parsing Fields");
					inst->pRunServer->State.eState = eBRB_RSSTATE_INIT_ERROR;
					inst->eStep = eSTEP_INIT;
					break;
				}
			}
			break;

		case eSTEP_FINISHED:
			inst->nStatus = 0;
			inst->pRunServer->State.eState = eBRB_RSSTATE_INIT_DONE;
			inst->eStep = eSTEP_INIT;
			break;

	}
}

// Wert aus dem Datenobjekt lesen
BOOL ParseServerValue(STRING** ppStart, STRING* pPar, STRING* pValue)
{
	BOOL bResult = 0;
	UDINT nLineLen = brsstrlen((UDINT)*ppStart);
	DINT nStartPar = BrbStringGetIndexOf(*ppStart, pPar, nLineLen);
	if(nStartPar > -1)
	{
		DINT nStartVal = nStartPar + (DINT)strlen(pPar);
		if(nStartVal >= 0)
		{
			DINT nEndVal = BrbStringGetIndexOf(*ppStart, ",", nLineLen);
			if(nEndVal > nStartVal)
			{
				// Bis zum nächsten Komma lesen
				UDINT nLen = (UDINT)(nEndVal- nStartVal);
				BrbStringGetSubText(*ppStart, (UDINT)nStartVal, nLen, pValue);
				BrbStringTrimLeft(pValue, " ");
				BrbStringTrimRight(pValue, " ");
				*ppStart += nEndVal+1;
				bResult = 1;
			}
			else if(nEndVal == -1)
			{
				// Kein Komma am Schluss -> Bis Ende lesen
				UDINT nLen = nLineLen - (UDINT)nStartVal;
				BrbStringGetSubText(*ppStart, (UDINT)nStartVal, nLen, pValue);
				BrbStringTrimLeft(pValue, " ");
				BrbStringTrimRight(pValue, " ");
				*ppStart += nEndVal+1;
				bResult = 1;
			}
		}
	}
	return bResult;
}

// NOLINTEND(readability-*, bugprone-easily-swappable-parameters, bugprone-branch-clone, clang-diagnostic-invalid-utf8, clang-diagnostic-invalid-source-encoding, clang-diagnostic-pointer-arith, clang-diagnostic-strict-prototypes, hicpp-uppercase-literal-suffix, cppcoreguidelines-*, performance-*)
```

#### BrbUaRunServerCyclic.c
```c
#include <bur/plctypes.h>
#ifdef __cplusplus
	extern "C"
	{
#endif

#include "BrbLibUa.h"
#include <string.h>
#include <AnsiCFunc.h>

#ifdef __cplusplus
	};
#endif

// NOLINTBEGIN(readability-*, bugprone-easily-swappable-parameters, bugprone-branch-clone, clang-diagnostic-invalid-utf8, clang-diagnostic-invalid-source-encoding, clang-diagnostic-pointer-arith, clang-diagnostic-strict-prototypes, hicpp-uppercase-literal-suffix, cppcoreguidelines-*, performance-*)

// Eigene Enums und Typen
enum Steps_ENUM
{
	eSTEP_INIT,
	eSTEP_GET_NAMESPACE,
	eSTEP_GET_EVENT_NS,
	eSTEP_GET_EVENT_FIELD_NS,
	eSTEP_RUNNING,
};

/* Behandelt eine Server-Instanz */
void BrbUaRunServerCyclic(struct BrbUaRunServerCyclic* inst)
{
	switch(inst->eStep)
	{
		case eSTEP_INIT:
			// Fub initialisieren
			inst->nStatus = eBRB_ERR_OK;
			//memset(&inst->fbUaSrv_GetServerState, 0, sizeof(inst->fbUaSrv_GetServerState));
			// Server-Pointer prüfen
			if(inst->pRunServer != 0)
			{
				inst->pRunServer->State.nErroId = 0;
				if(inst->pRunServer->State.eState == eBRB_RSSTATE_INIT_DONE)
				{
					inst->nNamespaceIndex = 0;
					inst->nEventIndex = 0;
					inst->nEventFieldIndex = 0;
					inst->eStep = eSTEP_GET_NAMESPACE;
				}
				else
				{
					inst->nStatus = eBRB_ERR_INVALID_PARAMETER;
					inst->pRunServer->State.nErroId = inst->nStatus;
					strcpy(inst->pRunServer->State.sErrorText, "Cyclic error: Init not done");
				}
			}
			else
			{
				inst->nStatus = eBRB_ERR_NULL_POINTER;
			}
			break;

		case eSTEP_GET_NAMESPACE:
			// NamespaceIndex ermitteln
			inst->pRunServer->State.eState = eBRB_RSSTATE_DETECTING;
			if(inst->pRunServer->Namespaces.nNamespaceCount > 0 && inst->pRunServer->Namespaces.pNamespaces != 0)
			{
				if(inst->nNamespaceIndex < inst->pRunServer->Namespaces.nNamespaceCount)
				{
					BrbUaRsNamespace_TYP* pNamespace = ((BrbUaRsNamespace_TYP*)inst->pRunServer->Namespaces.pNamespaces) + inst->nNamespaceIndex;
					inst->fbUaSrv_GetNamespaceIndex.Execute = 1;
					BrbStringCopy(inst->fbUaSrv_GetNamespaceIndex.NamespaceUri, pNamespace->sNamespaceUri, sizeof(inst->fbUaSrv_GetNamespaceIndex.NamespaceUri));
					if(inst->fbUaSrv_GetNamespaceIndex.Done == 1)
					{
						inst->fbUaSrv_GetNamespaceIndex.Execute = 0;
						pNamespace->nNamespaceIndex = inst->fbUaSrv_GetNamespaceIndex.NamespaceIndex;
						pNamespace->nErrorId = 0x00000000; // = Good
						inst->nNamespaceIndex += 1;
					}
					else if(inst->fbUaSrv_GetNamespaceIndex.Error == 1)
					{
						inst->fbUaSrv_GetNamespaceIndex.Execute = 0;
						pNamespace->nNamespaceIndex = 0;
						pNamespace->nErrorId = inst->fbUaSrv_GetNamespaceIndex.ErrorID;
						inst->pRunServer->State.nErroId = inst->fbUaSrv_GetNamespaceIndex.ErrorID;
						strcpy(inst->pRunServer->State.sErrorText, "Cyclic error on getting Namespace#");
						STRING sHelp[16];
						brsitoa(inst->nNamespaceIndex, (UDINT)&sHelp);
						BrbStringCat(inst->pRunServer->State.sErrorText, sHelp, sizeof(inst->pRunServer->State.sErrorText));
						inst->nNamespaceIndex += 1;
					}
				}
				else
				{
					inst->eStep = eSTEP_GET_EVENT_NS;
				}
			}
			else
			{
				// Keine Namespaces: Andere Eintragungen mache keinen Sinn
				inst->eStep = eSTEP_RUNNING;
			}
			break;

		case eSTEP_GET_EVENT_NS:
			// Bei allen Events den ServerNamespaceIndex eintragen (in 64-Blöcken)
			inst->pRunServer->State.eState = eBRB_RSSTATE_DETECTING;
			if(inst->pRunServer->Events.nEventCount > 0 && inst->pRunServer->Events.pEvents != 0)
			{
				DINT nRemainingItemsCount = inst->pRunServer->Events.nEventCount - inst->nEventIndex;
				if(nRemainingItemsCount > 0)
				{
					UINT nItemCount = (UINT)nRemainingItemsCount;
					if(nRemainingItemsCount > 64)
					{
						nItemCount = 64;
					}
					for(inst->nLoopIndex=0; inst->nLoopIndex < nItemCount; inst->nLoopIndex++)
					{
						// ServerNamespaceIndex aus geparsten DatObj-Index für jedes Event ermitteln
						BrbUaRsEventIntern_TYP* pEvent = ((BrbUaRsEventIntern_TYP*)inst->pRunServer->Events.pEvents) + inst->nEventIndex + inst->nLoopIndex;
						pEvent->TypeNodeId.NamespaceIndex = BrbUaRsGetNamespace(inst->pRunServer, pEvent->nDatObjNamespaceIndex, 0);
					}
					inst->nEventIndex += nItemCount;
				}
				else
				{
					inst->nEventIndex = 0;
					inst->eStep = eSTEP_GET_EVENT_FIELD_NS;
				}
			}
			else
			{
				inst->eStep = eSTEP_RUNNING;
			}
			break;

		case eSTEP_GET_EVENT_FIELD_NS:
			// Bei allen EventFields den ServerNamespaceIndex eintragen (in 4-Blöcken)
			if(inst->pRunServer->Events.nEventCount > 0 && inst->pRunServer->Events.pEvents != 0)
			{
				// Events und deren Fields durchtickern
				UINT nEventFieldLoopCount = 0;
				BOOL bLeaveEventLoop = 0;
				do
				{
					if(inst->nEventIndex < inst->pRunServer->Events.nEventCount)
					{
						BrbUaRsEventIntern_TYP* pEvent = ((BrbUaRsEventIntern_TYP*)inst->pRunServer->Events.pEvents) + inst->nEventIndex;
						if(inst->nEventFieldIndex < pEvent->nFieldCount)
						{
							// ServerNamespaceIndex in jedem Element des Browse-Pfads ermitteln und austauschen
							UaSrv_FireEventFieldType* pEventField = ((UaSrv_FireEventFieldType*)pEvent->pFields) + inst->nEventFieldIndex;
							nEventFieldLoopCount += 1;
							UDINT nPathLen = brsstrlen((UDINT)&pEventField->BrowsePath);
							UINT nOffset = 0;
							BOOL bLeaveBrowsePathLoop = 0;
							do
							{
								// BrowsePath durchtickern
								if(nOffset < nPathLen)
								{
									// Nach / suchen
									DINT nStart = BrbStringGetIndexOf((STRING*)&pEventField->BrowsePath + nOffset, "/", 0);
									if(nStart > -1)
									{
										// Nach : suchen
										DINT nEnd = BrbStringGetIndexOf((STRING*)&pEventField->BrowsePath + nOffset + nStart + 1, ":", 0);
										if(nEnd > nStart)
										{
											// Zwischen / und : könnte ein NamespaceIndex liegen
											DINT nLen = nEnd - nStart;
											if(nLen > 0)
											{
												// Vermutlichen NamespaceIndex ermitteln
												STRING sOldNamespaceIndex[nLen+1];
												BrbStringGetSubTextByLen((STRING*)&pEventField->BrowsePath + nOffset + nStart + 1, (UDINT)nLen, (STRING*)&sOldNamespaceIndex);
												// Auf Nummer prüfen
												if(BrbStringIsNumerical(sOldNamespaceIndex) == 1)
												{
													// NamespaceIndex vorhanden
													UINT nOldNamespaceIndex = (UINT)BrbAsciiToUdint((STRING*)&sOldNamespaceIndex);
													UINT nNewNamespaceIndex = BrbUaRsGetNamespace(inst->pRunServer, nOldNamespaceIndex, 0);
													// Auf Unterschied prüfen
													if(nNewNamespaceIndex != nOldNamespaceIndex)
													{
														// Alten NamespaceIndex rausschneiden
														BrbStringCut((STRING*)&pEventField->BrowsePath + nOffset, (UDINT)nStart + 1, (UDINT)nLen, 0);
														// Neuen NamespaceIndex einfügen
														STRING sNewNamespaceIndex[12];
														brsitoa((DINT)nNewNamespaceIndex, (UDINT)&sNewNamespaceIndex);
														BrbStringInsert((STRING*)&pEventField->BrowsePath + nOffset, (UDINT)nStart + 1, (STRING*)sNewNamespaceIndex);
													}
												}
											}
											nOffset += nEnd;
										}
										else
										{
											inst->nEventFieldIndex += 1;
											bLeaveBrowsePathLoop = 1;
										}
									}
									else
									{
										inst->nEventFieldIndex += 1;
										bLeaveBrowsePathLoop = 1;
									}
								}
								else
								{
									inst->nEventFieldIndex += 1;
									bLeaveBrowsePathLoop = 1;
								}
							} while(bLeaveBrowsePathLoop == 0);
							if(nEventFieldLoopCount >= 4)
							{
								nEventFieldLoopCount = 0;
								bLeaveEventLoop = 1;
							}
						}
						else
						{
							// Nächstes Event
							inst->nEventFieldIndex = 0;
							inst->nEventIndex += 1;
						}
					}
					else
					{
						// Alle Events behandelt
						bLeaveEventLoop = 1;
						inst->eStep = eSTEP_RUNNING;
					}
				} while(bLeaveEventLoop == 0);
			}
			else
			{
				// Keine Events
				inst->eStep = eSTEP_RUNNING;
			}
			break;

		case eSTEP_RUNNING:
			inst->pRunServer->State.eState = eBRB_RSSTATE_RUNNING;
			// Server-Status abfragen
			inst->pRunServer->State.eServerState = UaSrv_GetServerState();
			break;

	}

	// Aufruf aller FB's
	UaSrv_GetNamespaceIndex(&inst->fbUaSrv_GetNamespaceIndex);
}

// NOLINTEND(readability-*, bugprone-easily-swappable-parameters, bugprone-branch-clone, clang-diagnostic-invalid-utf8, clang-diagnostic-invalid-source-encoding, clang-diagnostic-pointer-arith, clang-diagnostic-strict-prototypes, hicpp-uppercase-literal-suffix, cppcoreguidelines-*, performance-*)
```

#### BrbUaRunServerExit.c
```c
#include <bur/plctypes.h>
#ifdef __cplusplus
	extern "C"
	{
#endif

#include "BrbLibUa.h"
#include <string.h>
#include <AnsiCFunc.h>

#ifdef __cplusplus
	};
#endif

// NOLINTBEGIN(readability-*, bugprone-easily-swappable-parameters, bugprone-branch-clone, clang-diagnostic-invalid-utf8, clang-diagnostic-invalid-source-encoding, clang-diagnostic-pointer-arith, clang-diagnostic-strict-prototypes, hicpp-uppercase-literal-suffix, cppcoreguidelines-*, performance-*)

// Eigene Enums und Typen
enum Steps_ENUM
{
	eSTEP_INIT,
	eSTEP_FREE_EVENTS,
	eSTEP_FINISHED,
};

/* Exilisiert eine Client-Instanz */
void BrbUaRunServerExit(struct BrbUaRunServerExit* inst)
{
	switch(inst->eStep)
	{
		case eSTEP_INIT:
			// Fub initialisieren
			inst->nStatus =  eBRB_ERR_BUSY;
			// Client-Pointer prüfen
			if(inst->pRunServer != 0)
			{
				inst->pRunServer->State.eState = eBRB_RSSTATE_EXITING;
				inst->pRunServer->State.nErroId = 0x00000000;
				strcpy(inst->pRunServer->State.sErrorText, "");
				inst->nEventIndex = 0;
				inst->eStep = eSTEP_FREE_EVENTS;
			}
			else
			{
				inst->nStatus = eBRB_ERR_NULL_POINTER;
				inst->eStep = eSTEP_INIT;
			}
			break;

		case eSTEP_FREE_EVENTS:
			// Speicher für alle Events freigeben
			inst->nStatus  = eBRB_ERR_BUSY;
			if(inst->pRunServer->Events.nEventCount > 0 && inst->pRunServer->Events.pEvents != 0 && inst->pRunServer->Events.nMemLen > 0)
			{
				inst->nFreeStatus = TMP_free(inst->pRunServer->Events.nMemLen, (void*)inst->pRunServer->Events.pEvents);
				if(inst->nFreeStatus == 0)
				{
					inst->pRunServer->Events.nEventCount = 0;
					inst->pRunServer->Events.pEvents = 0;
					inst->pRunServer->Events.nMemLen = 0;
					inst->eStep = eSTEP_FINISHED;
				}
				else
				{
					// Fehler
					inst->nStatus = inst->nFreeStatus;
					inst->pRunServer->State.nErroId = inst->nStatus;
					strcpy(inst->pRunServer->State.sErrorText, "Exit error on freeing memory for events");
					inst->pRunServer->State.eState = eBRB_RSSTATE_EXIT_ERROR;
					inst->eStep = eSTEP_INIT;
				}
			}
			else
			{
				// Keine Events angegeben
				inst->eStep = eSTEP_FINISHED;
			}
			break;

		case eSTEP_FINISHED:
			inst->nStatus = 0;
			inst->pRunServer->State.eState = eBRB_RSSTATE_EXIT_DONE;
			inst->eStep = eSTEP_INIT;
			break;

	}

}

// NOLINTEND(readability-*, bugprone-easily-swappable-parameters, bugprone-branch-clone, clang-diagnostic-invalid-utf8, clang-diagnostic-invalid-source-encoding, clang-diagnostic-pointer-arith, clang-diagnostic-strict-prototypes, hicpp-uppercase-literal-suffix, cppcoreguidelines-*, performance-*)
```

#### BrbUaRsFireEvent.c
```c
#include <bur/plctypes.h>
#ifdef __cplusplus
	extern "C"
	{
#endif

#include "BrbLibUa.h"
#include <string.h>
#include <AnsiCFunc.h>

#ifdef __cplusplus
	};
#endif

// NOLINTBEGIN(readability-*, bugprone-easily-swappable-parameters, bugprone-branch-clone, clang-diagnostic-invalid-utf8, clang-diagnostic-invalid-source-encoding, clang-diagnostic-pointer-arith, clang-diagnostic-strict-prototypes, hicpp-uppercase-literal-suffix, cppcoreguidelines-*, performance-*)

// Eigene Enums und Typen
enum Steps_ENUM
{
	eSTEP_INIT,
	eSTEP_FIRE,
	eSTEP_FIRE_WAIT,
};

/* Liest eine WriteBlock vom Server */
void BrbUaRsFireEvent(struct BrbUaRsFireEvent* inst)
{
	switch(inst->eStep)
	{
		case eSTEP_INIT:
			// Fub initialisieren
			inst->nStatus =  eBRB_ERR_BUSY;
			inst->nErrorId = 0x00000000; // Good
			BrbUaGetStatusCodeText(inst->nErrorId, inst->sErrorId, sizeof(inst->nErrorId));
			memset(&inst->fbUaSrv_FireEvent, 0, sizeof(inst->fbUaSrv_FireEvent));
			inst->bInit = 0;
			// Parameter prüfen
			if(inst->pRunServer != 0)
			{
				if(inst->pRunServer->State.eState == eBRB_RSSTATE_RUNNING)
				{
					if(inst->pRunServer->Events.nEventCount > 0 && inst->pRunServer->Events.pEvents != 0)
					{
						if(inst->nEventIndex < inst->pRunServer->Events.nEventCount)
						{
							inst->bInit = 1;
							inst->eStep = eSTEP_FIRE;
						}
						else
						{
							inst->nStatus = eBRB_ERR_UA_INVALID_INDEX;
						}
					}
					else
					{
						inst->nStatus = eBRB_ERR_UA_NO_ELEMENTS;
					}
				}
				else
				{
					inst->nStatus = eBRB_ERR_UA_NOT_RUNNING;
				}
			}
			else
			{
				inst->nStatus = eBRB_ERR_NULL_POINTER;
			}
			break;

		case eSTEP_FIRE:
			// Event feuern
			inst->nStatus  = eBRB_ERR_BUSY;
			inst->bInit = 0;
			{
				BrbUaRsEventIntern_TYP* pEvent = (((BrbUaRsEventIntern_TYP*)inst->pRunServer->Events.pEvents)  + inst->nEventIndex);
				inst->fbUaSrv_FireEvent.Execute = 1;
				memcpy(&inst->fbUaSrv_FireEvent.EventType, &pEvent->TypeNodeId, sizeof(UANodeID));
				inst->fbUaSrv_FireEvent.EventFieldCount = pEvent->nFieldCount;
				inst->fbUaSrv_FireEvent.EventFields = (void*)pEvent->pFields;
			}
			inst->eStep = eSTEP_FIRE_WAIT;
			break;

		case eSTEP_FIRE_WAIT:
			// Warten, bis Block gelesen wurde
			inst->nStatus  = eBRB_ERR_BUSY;
			if(inst->fbUaSrv_FireEvent.Done == 1)
			{
				inst->fbUaSrv_FireEvent.Execute = 0;
				inst->nStatus  = eBRB_ERR_OK;
				inst->nErrorId = inst->fbUaSrv_FireEvent.ErrorID;
				BrbUaGetStatusCodeText(inst->nErrorId, inst->sErrorId, sizeof(inst->nErrorId));
				inst->nFireCount++;
				inst->eStep = eSTEP_INIT;
			}
			else if(inst->fbUaSrv_FireEvent.Error == 1)
			{
				inst->fbUaSrv_FireEvent.Execute = 0;
				inst->nStatus  = eBRB_ERR_UA_ERROR;
				inst->nErrorId = inst->fbUaSrv_FireEvent.ErrorID;
				if(inst->nErrorId == 0)
				{
					// Fehler trat bei einem Field auf
					BrbUaRsEventIntern_TYP* pEvent = (((BrbUaRsEventIntern_TYP*)inst->pRunServer->Events.pEvents)  + inst->nEventIndex);
					UINT nEventFieldIndex = 0;
					for(nEventFieldIndex=0; nEventFieldIndex<pEvent->nFieldCount; nEventFieldIndex++)
					{
						UaSrv_FireEventFieldType* pEventField = ((UaSrv_FireEventFieldType*)pEvent->pFields) + nEventFieldIndex;
						if(pEventField->ErrorID != 0)
						{
							inst->nErrorId = pEventField->ErrorID;
							break;
						}
					}
				}
				BrbUaGetStatusCodeText(inst->nErrorId, inst->sErrorId, sizeof(inst->nErrorId));
				inst->eStep = eSTEP_INIT;
			}
			break;

	}

	// Aufruf aller FB's
	UaSrv_FireEvent(&inst->fbUaSrv_FireEvent);
}

// NOLINTEND(readability-*, bugprone-easily-swappable-parameters, bugprone-branch-clone, clang-diagnostic-invalid-utf8, clang-diagnostic-invalid-source-encoding, clang-diagnostic-pointer-arith, clang-diagnostic-strict-prototypes, hicpp-uppercase-literal-suffix, cppcoreguidelines-*, performance-*)
```

#### BrbUaRsGetNamespace.c
```c
#include <bur/plctypes.h>
#ifdef __cplusplus
	extern "C"
	{
#endif

#include "BrbLibUa.h"
#include <string.h>
#include <AnsiCFunc.h>

#ifdef __cplusplus
	};
#endif

// NOLINTBEGIN(readability-*, bugprone-easily-swappable-parameters, bugprone-branch-clone, clang-diagnostic-invalid-utf8, clang-diagnostic-invalid-source-encoding, clang-diagnostic-pointer-arith, clang-diagnostic-strict-prototypes, hicpp-uppercase-literal-suffix, cppcoreguidelines-*, performance-*)

/* Gibt den Server-Namespace aufgrund des DataObjekt-NamespaceIndex zurück */
unsigned short BrbUaRsGetNamespace(struct BrbUaRunServer_TYP* pRunServer, unsigned short nDatObjNamespaceIndex, struct BrbUaRsNamespace_TYP* pServerNamespace)
{
	UINT nServerNamespaceIndex = 0;
	if(pRunServer != 0)
	{
		if(pRunServer->Namespaces.nNamespaceCount > 0 && pRunServer->Namespaces.pNamespaces != 0)
		{
			if(nDatObjNamespaceIndex < pRunServer->Namespaces.nNamespaceCount)
			{
				BrbUaRsNamespace_TYP* pNamespace = ((BrbUaRsNamespace_TYP*)pRunServer->Namespaces.pNamespaces) + nDatObjNamespaceIndex;
				nServerNamespaceIndex = pNamespace->nNamespaceIndex;
				if(pServerNamespace != 0)
				{
					memcpy(pServerNamespace, (USINT*)(((BrbUaRsNamespace_TYP*)pRunServer->Namespaces.pNamespaces) + nDatObjNamespaceIndex), sizeof(BrbUaRsNamespace_TYP));
				}
			}
		}
	}
	return nServerNamespaceIndex;
}

// NOLINTEND(readability-*, bugprone-easily-swappable-parameters, bugprone-branch-clone, clang-diagnostic-invalid-utf8, clang-diagnostic-invalid-source-encoding, clang-diagnostic-pointer-arith, clang-diagnostic-strict-prototypes, hicpp-uppercase-literal-suffix, cppcoreguidelines-*, performance-*)
```
